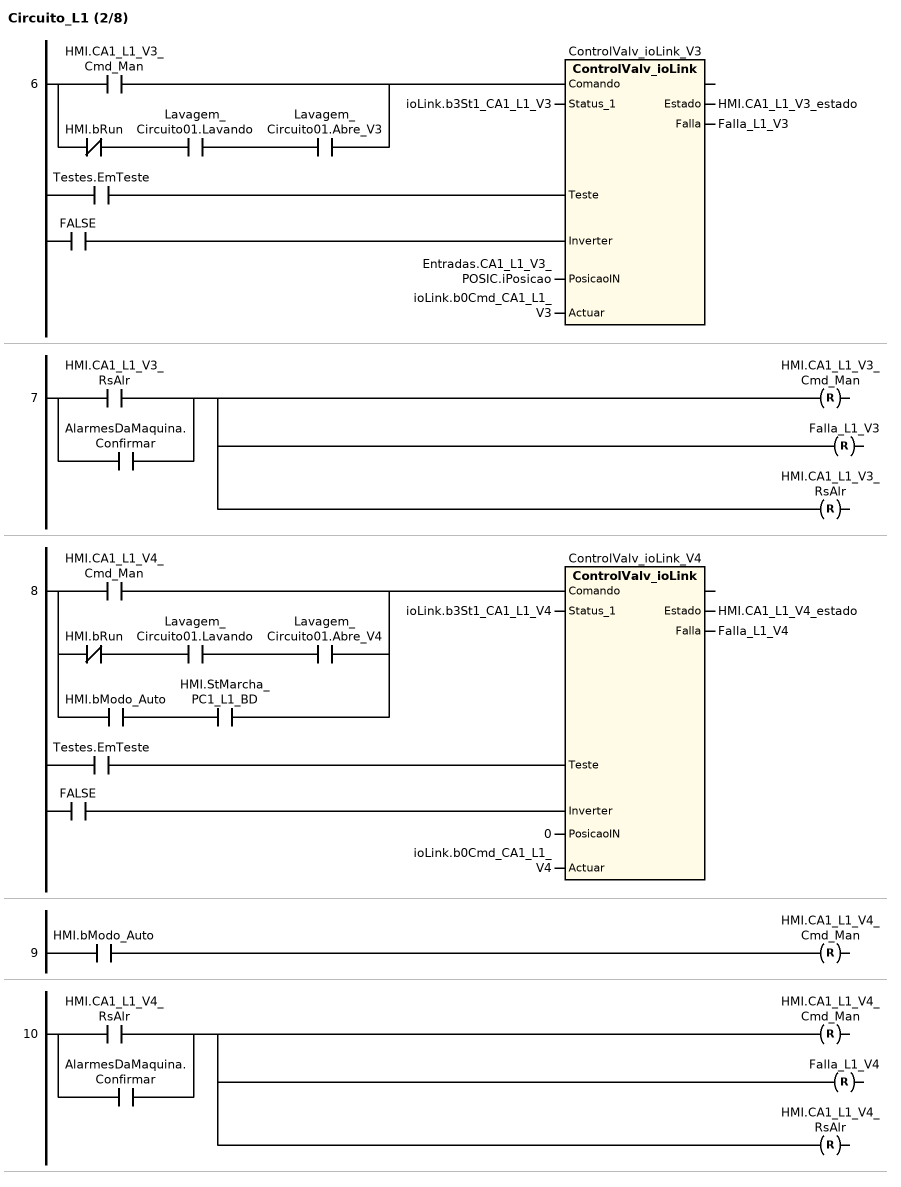
// NETWORK 6
ControlValv_ioLink_V3(
    Comando := HMI.CA1_L1_V3_Cmd_Man OR NOT HMI.bRun AND Lavagem_Circuito01.Lavando AND Lavagem_Circuito01.Abre_V3,
    Status_1 := ioLink.b3St1_CA1_L1_V3,
    Teste := Testes.EmTeste,
    Inverter := FALSE,
    PosicaoIN := Entradas.CA1_L1_V3_POSIC.iPosicao,
    Actuar := ioLink.b0Cmd_CA1_L1_V3,
    Estado => HMI.CA1_L1_V3_estado,
    Falla => Falla_L1_V3); // ControlValv_ioLink

// NETWORK 7
_w3 := HMI.CA1_L1_V3_RsAlr OR AlarmesDaMaquina.Confirmar;
HMI.CA1_L1_V3_Cmd_Man R= _w3;
Falla_L1_V3 R= _w3;
HMI.CA1_L1_V3_RsAlr R= _w3;

// NETWORK 8
ControlValv_ioLink_V4(
    Comando := HMI.CA1_L1_V4_Cmd_Man OR NOT HMI.bRun AND Lavagem_Circuito01.Lavando AND Lavagem_Circuito01.Abre_V4 OR HMI.bModo_Auto AND HMI.StMarcha_PC1_L1_BD,
    Status_1 := ioLink.b3St1_CA1_L1_V4,
    Teste := Testes.EmTeste,
    Inverter := FALSE,
    PosicaoIN := 0,
    Actuar := ioLink.b0Cmd_CA1_L1_V4,
    Estado => HMI.CA1_L1_V4_estado,
    Falla => Falla_L1_V4); // ControlValv_ioLink

// NETWORK 9
HMI.CA1_L1_V4_Cmd_Man R= HMI.bModo_Auto;

// NETWORK 10
_w4 := HMI.CA1_L1_V4_RsAlr OR AlarmesDaMaquina.Confirmar;
HMI.CA1_L1_V4_Cmd_Man R= _w4;
Falla_L1_V4 R= _w4;
HMI.CA1_L1_V4_RsAlr R= _w4;

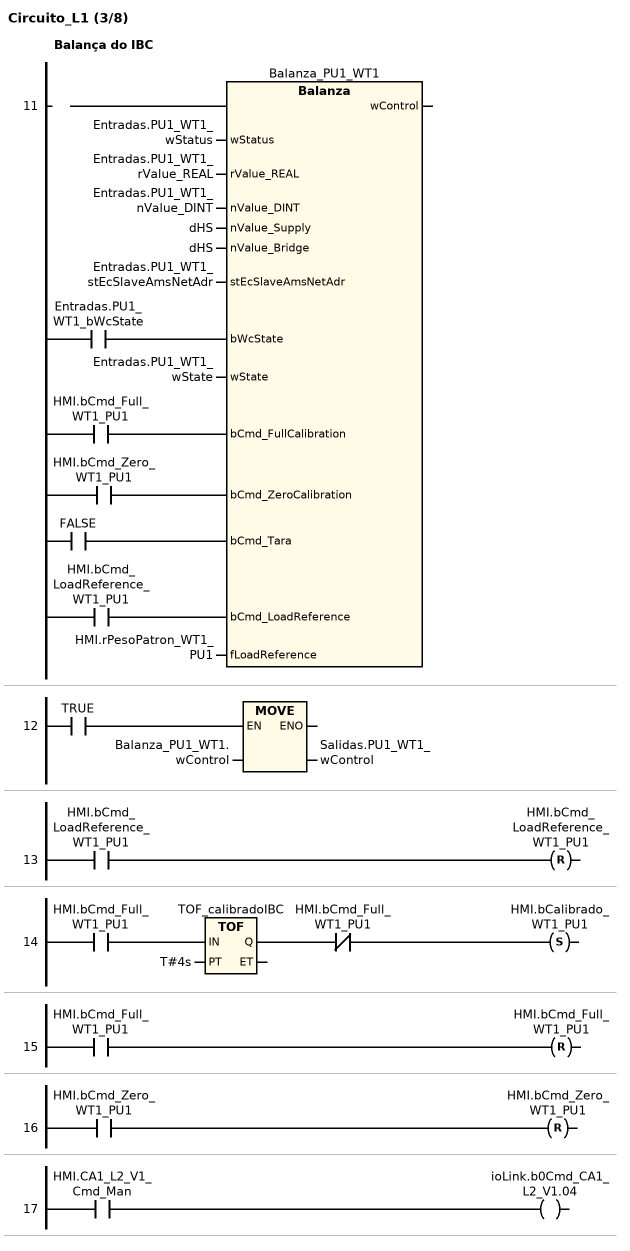
// NETWORK 11: Balança do IBC
Balanza_PU1_WT1(
    wStatus := Entradas.PU1_WT1_wStatus,
    rValue_REAL := Entradas.PU1_WT1_rValue_REAL,
    nValue_DINT := Entradas.PU1_WT1_nValue_DINT,
    nValue_Supply := dHS,
    nValue_Bridge := dHS,
    stEcSlaveAmsNetAdr := Entradas.PU1_WT1_stEcSlaveAmsNetAdr,
    bWcState := Entradas.PU1_WT1_bWcState,
    wState := Entradas.PU1_WT1_wState,
    bCmd_FullCalibration := HMI.bCmd_Full_WT1_PU1,
    bCmd_ZeroCalibration := HMI.bCmd_Zero_WT1_PU1,
    bCmd_Tara := FALSE,
    bCmd_LoadReference := HMI.bCmd_LoadReference_WT1_PU1,
    fLoadReference := HMI.rPesoPatron_WT1_PU1); // Balanza

// NETWORK 12
Salidas.PU1_WT1_wControl := Balanza_PU1_WT1.wControl;

// NETWORK 13
HMI.bCmd_LoadReference_WT1_PU1 R= HMI.bCmd_LoadReference_WT1_PU1;

// NETWORK 14
TOF_calibradoIBC(IN := HMI.bCmd_Full_WT1_PU1, PT := T#4s); // TOF
HMI.bCalibrado_WT1_PU1 S= TOF_calibradoIBC.Q AND NOT HMI.bCmd_Full_WT1_PU1;

// NETWORK 15
HMI.bCmd_Full_WT1_PU1 R= HMI.bCmd_Full_WT1_PU1;

// NETWORK 16
HMI.bCmd_Zero_WT1_PU1 R= HMI.bCmd_Zero_WT1_PU1;

// NETWORK 17
ioLink.b0Cmd_CA1_L2_V1.04 := HMI.CA1_L2_V1_Cmd_Man;

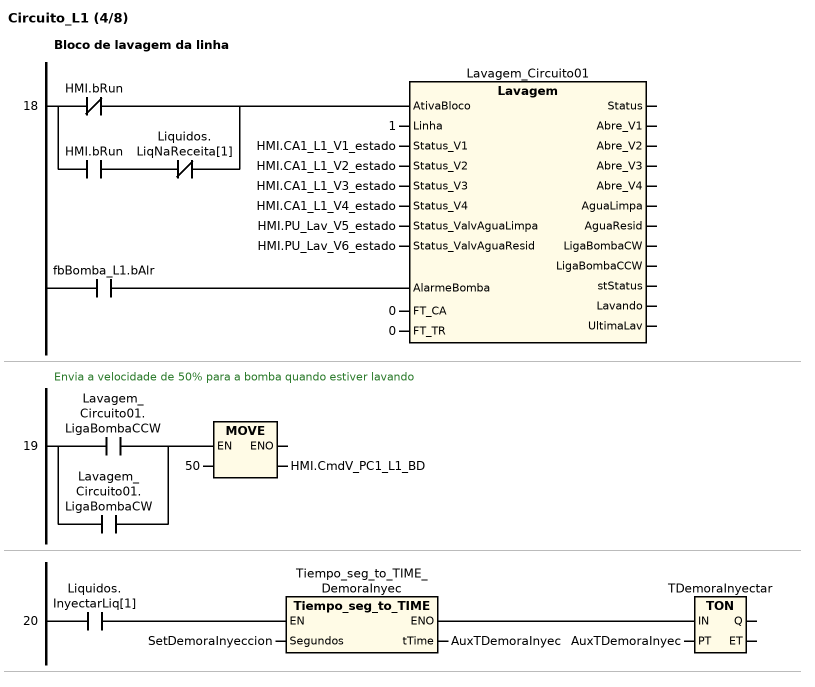
// NETWORK 18: Bloco de lavagem da linha
Lavagem_Circuito01(
    AtivaBloco := NOT HMI.bRun OR HMI.bRun AND NOT Liquidos.LiqNaReceita[1],
    Linha := 1,
    Status_V1 := HMI.CA1_L1_V1_estado,
    Status_V2 := HMI.CA1_L1_V2_estado,
    Status_V3 := HMI.CA1_L1_V3_estado,
    Status_V4 := HMI.CA1_L1_V4_estado,
    Status_ValvAguaLimpa := HMI.PU_Lav_V5_estado,
    Status_ValvAguaResid := HMI.PU_Lav_V6_estado,
    AlarmeBomba := fbBomba_L1.bAlr,
    FT_CA := 0,
    FT_TR := 0); // Lavagem

// NETWORK 19
// Envia a velocidade de 50% para a bomba quando estiver lavando
IF Lavagem_Circuito01.LigaBombaCCW OR Lavagem_Circuito01.LigaBombaCW THEN HMI.CmdV_PC1_L1_BD := 50; END_IF

// NETWORK 20
_w5 := Liquidos.InyectarLiq[1];
IF _w5 THEN
    Tiempo_seg_to_TIME_DemoraInyec(Segundos := SetDemoraInyeccion, tTime => AuxTDemoraInyec); // Tiempo_seg_to_TIME
END_IF
TDemoraInyectar(IN := _w5, PT := AuxTDemoraInyec); // TON

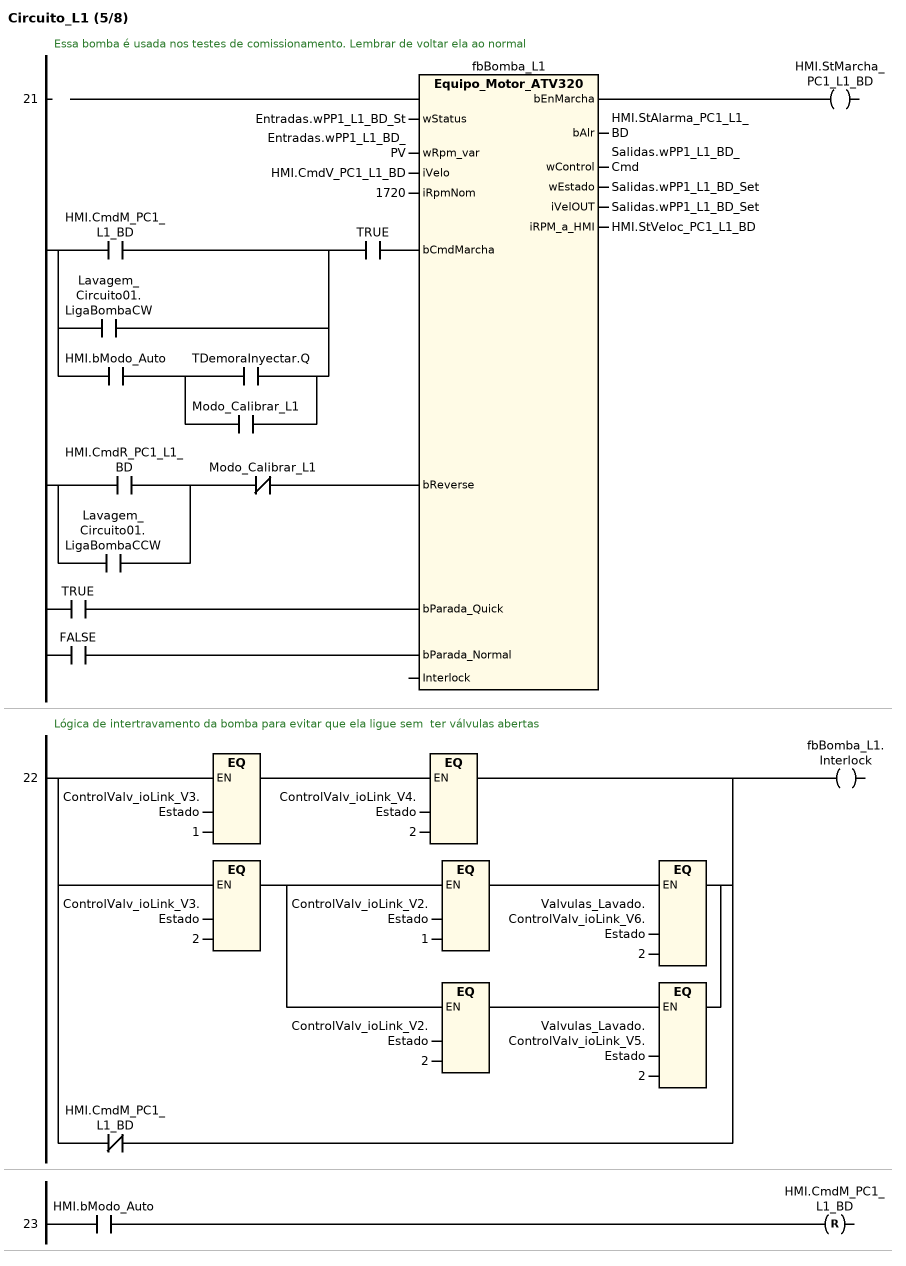
// NETWORK 21
// Essa bomba é usada nos testes de comissionamento. Lembrar de voltar ela ao normal
fbBomba_L1(
    wStatus := Entradas.wPP1_L1_BD_St,
    wRpm_var := Entradas.wPP1_L1_BD_PV,
    iVelo := HMI.CmdV_PC1_L1_BD,
    iRpmNom := 1720,
    bCmdMarcha := (HMI.CmdM_PC1_L1_BD OR Lavagem_Circuito01.LigaBombaCW OR HMI.bModo_Auto AND (TDemoraInyectar.Q OR Modo_Calibrar_L1)) AND TRUE,
    bReverse := (HMI.CmdR_PC1_L1_BD OR Lavagem_Circuito01.LigaBombaCCW) AND NOT Modo_Calibrar_L1,
    bParada_Quick := TRUE,
    bParada_Normal := FALSE,
    bAlr => HMI.StAlarma_PC1_L1_BD,
    wControl => Salidas.wPP1_L1_BD_Cmd,
    wEstado => Salidas.wPP1_L1_BD_Set,
    iVelOUT => Salidas.wPP1_L1_BD_Set,
    iRPM_a_HMI => HMI.StVeloc_PC1_L1_BD); // Equipo_Motor_ATV320
HMI.StMarcha_PC1_L1_BD := fbBomba_L1.bEnMarcha;

// NETWORK 22
// Lógica de intertravamento da bomba para evitar que ela ligue sem  ter válvulas abertas
_w6 := NOT HMI.CmdM_PC1_L1_BD;
IF NOT _w6 THEN
    _w7 := ControlValv_ioLink_V3.Estado = 2;
    _w6 := ControlValv_ioLink_V3.Estado = 1 AND ControlValv_ioLink_V4.Estado = 2 OR (_w7 AND ControlValv_ioLink_V2.Estado = 1 AND Valvulas_Lavado.ControlValv_ioLink_V6.Estado = 2 OR _w7 AND ControlValv_ioLink_V2.Estado = 2 AND Valvulas_Lavado.ControlValv_ioLink_V5.Estado = 2);
END_IF
fbBomba_L1.Interlock := _w6;

// NETWORK 23
HMI.CmdM_PC1_L1_BD R= HMI.bModo_Auto;

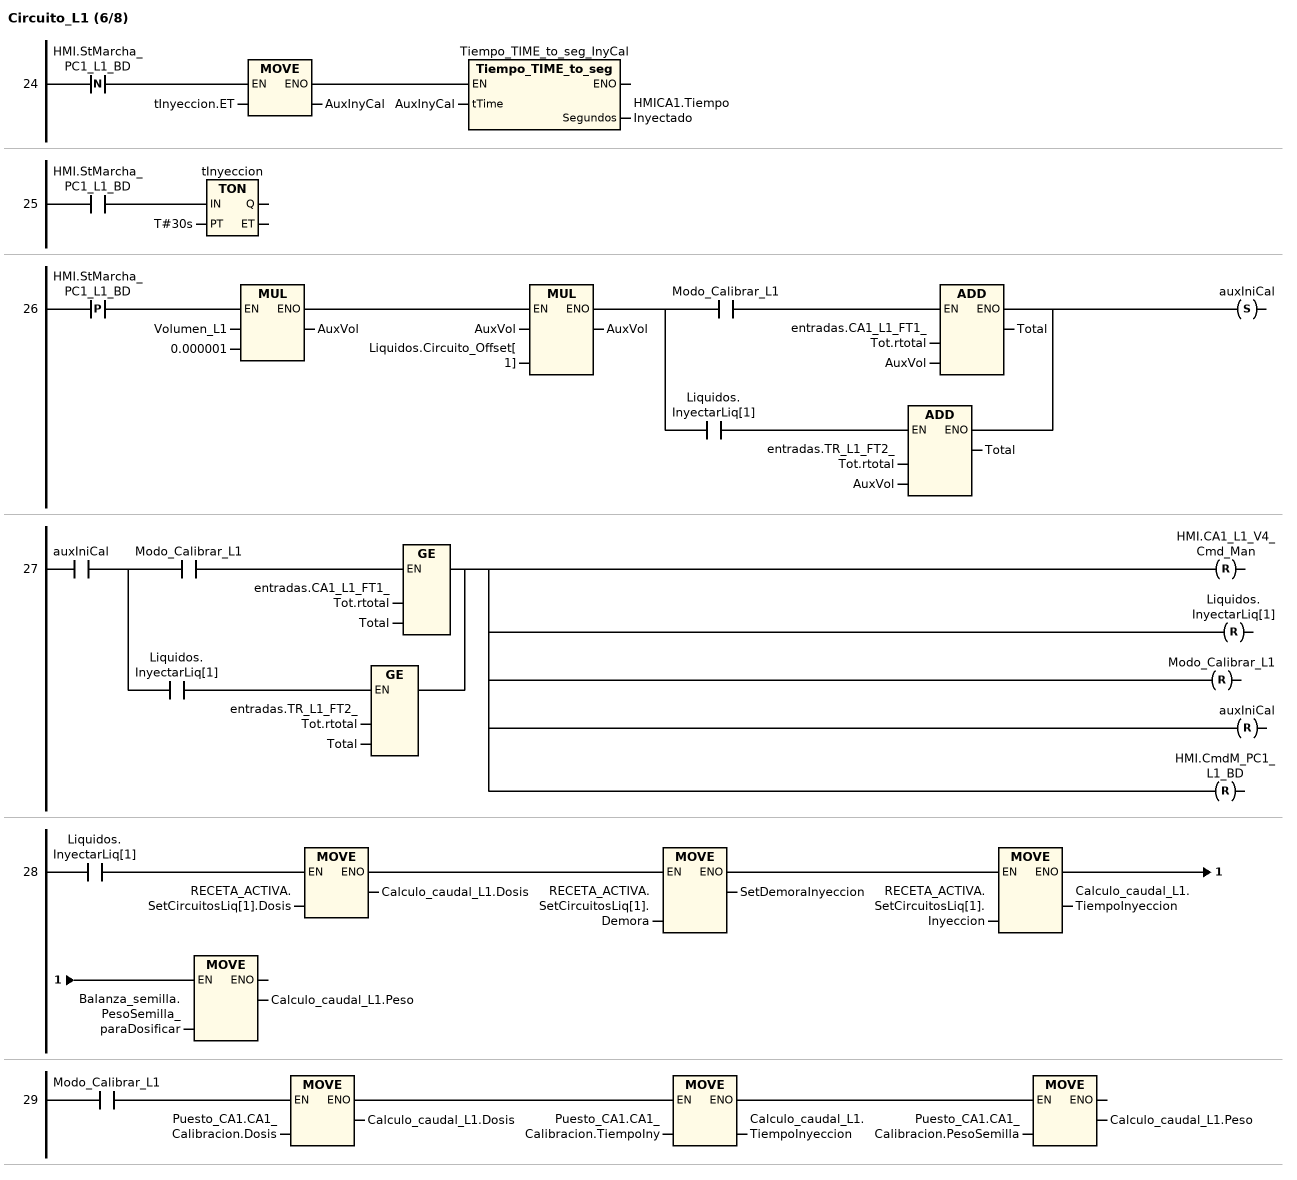
// NETWORK 24
_ft1(CLK := HMI.StMarcha_PC1_L1_BD);
_w8 := _ft1.Q;
IF _w8 THEN AuxInyCal := tInyeccion.ET; END_IF
IF _w8 THEN
    Tiempo_TIME_to_seg_InyCal(tTime := AuxInyCal, Segundos => HMICA1.TiempoInyectado); // Tiempo_TIME_to_seg
END_IF

// NETWORK 25
tInyeccion(IN := HMI.StMarcha_PC1_L1_BD, PT := T#30s); // TON

// NETWORK 26
_rt1(CLK := HMI.StMarcha_PC1_L1_BD);
_w9 := _rt1.Q;
IF _w9 THEN AuxVol := Volumen_L1 * 0.000001; END_IF
IF _w9 THEN AuxVol := AuxVol * Liquidos.Circuito_Offset[1]; END_IF
IF _w9 AND Modo_Calibrar_L1 THEN Total := entradas.CA1_L1_FT1_Tot.rtotal + AuxVol; END_IF
IF _w9 AND Liquidos.InyectarLiq[1] THEN Total := entradas.TR_L1_FT2_Tot.rtotal + AuxVol; END_IF
auxIniCal S= _w9 AND Modo_Calibrar_L1 OR _w9 AND Liquidos.InyectarLiq[1];

// NETWORK 27
_w10 := auxIniCal AND Modo_Calibrar_L1 AND entradas.CA1_L1_FT1_Tot.rtotal >= Total OR auxIniCal AND Liquidos.InyectarLiq[1] AND entradas.TR_L1_FT2_Tot.rtotal >= Total;
HMI.CA1_L1_V4_Cmd_Man R= _w10;
Liquidos.InyectarLiq[1] R= _w10;
Modo_Calibrar_L1 R= _w10;
auxIniCal R= _w10;
HMI.CmdM_PC1_L1_BD R= _w10;

// NETWORK 28
_w11 := Liquidos.InyectarLiq[1];
IF _w11 THEN Calculo_caudal_L1.Dosis := RECETA_ACTIVA.SetCircuitosLiq[1].Dosis; END_IF
IF _w11 THEN SetDemoraInyeccion := RECETA_ACTIVA.SetCircuitosLiq[1].Demora; END_IF
IF _w11 THEN Calculo_caudal_L1.TiempoInyeccion := RECETA_ACTIVA.SetCircuitosLiq[1].Inyeccion; END_IF
IF _w11 THEN Calculo_caudal_L1.Peso := Balanza_semilla.PesoSemilla_paraDosificar; END_IF

// NETWORK 29
_w12 := Modo_Calibrar_L1;
IF _w12 THEN Calculo_caudal_L1.Dosis := Puesto_CA1.CA1_Calibracion.Dosis; END_IF
IF _w12 THEN Calculo_caudal_L1.TiempoInyeccion := Puesto_CA1.CA1_Calibracion.TiempoIny; END_IF
IF _w12 THEN Calculo_caudal_L1.Peso := Puesto_CA1.CA1_Calibracion.PesoSemilla; END_IF

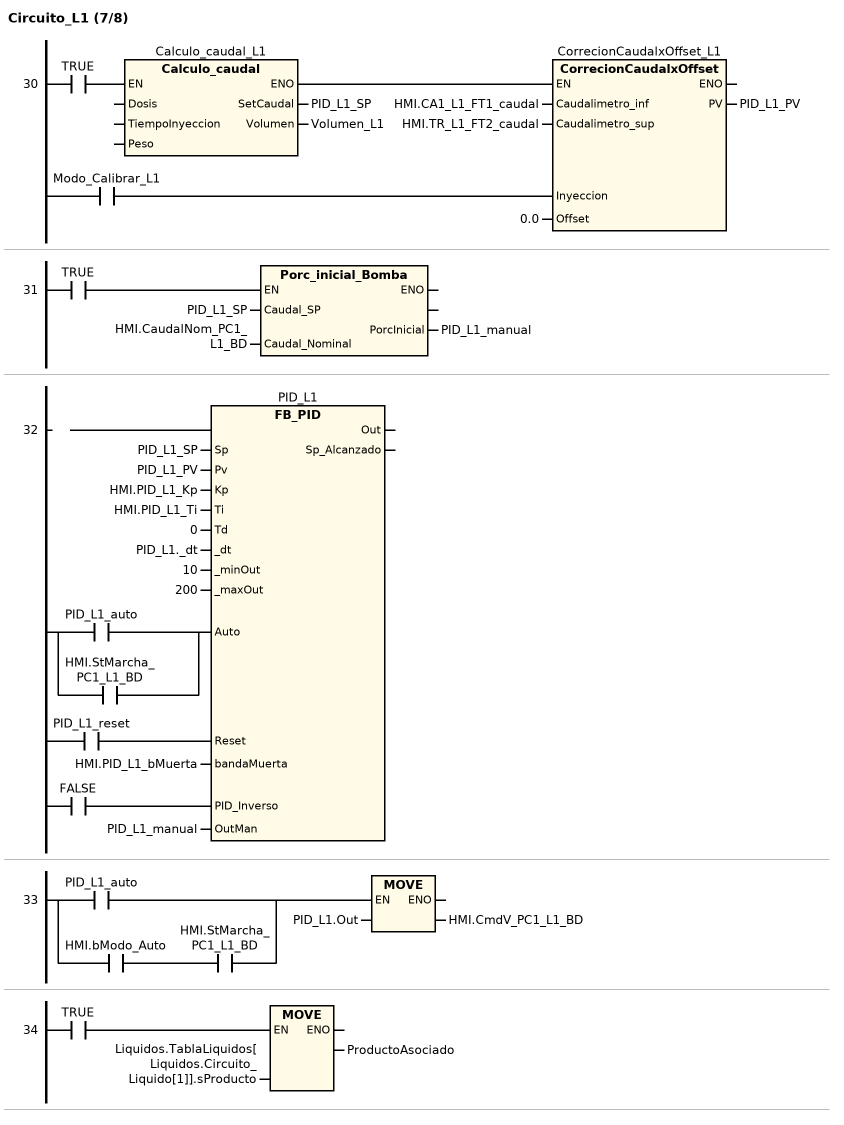
// NETWORK 30
Calculo_caudal_L1(SetCaudal => PID_L1_SP, Volumen => Volumen_L1); // Calculo_caudal
CorrecionCaudalxOffset_L1(
    Caudalimetro_inf := HMI.CA1_L1_FT1_caudal,
    Caudalimetro_sup := HMI.TR_L1_FT2_caudal,
    Inyeccion := Modo_Calibrar_L1,
    Offset := 0.0,
    PV => PID_L1_PV); // CorrecionCaudalxOffset

// NETWORK 31
Porc_inicial_Bomba(Caudal_SP := PID_L1_SP, Caudal_Nominal := HMI.CaudalNom_PC1_L1_BD, PorcInicial => PID_L1_manual);

// NETWORK 32
PID_L1(
    Sp := PID_L1_SP,
    Pv := PID_L1_PV,
    Kp := HMI.PID_L1_Kp,
    Ti := HMI.PID_L1_Ti,
    Td := 0,
    _dt := PID_L1._dt,
    _minOut := 10,
    _maxOut := 200,
    Auto := PID_L1_auto OR HMI.StMarcha_PC1_L1_BD,
    Reset := PID_L1_reset,
    bandaMuerta := HMI.PID_L1_bMuerta,
    PID_Inverso := FALSE,
    OutMan := PID_L1_manual); // FB_PID

// NETWORK 33
IF PID_L1_auto OR HMI.bModo_Auto AND HMI.StMarcha_PC1_L1_BD THEN HMI.CmdV_PC1_L1_BD := PID_L1.Out; END_IF

// NETWORK 34
ProductoAsociado := Liquidos.TablaLiquidos[Liquidos.Circuito_Liquido[1]].sProducto;

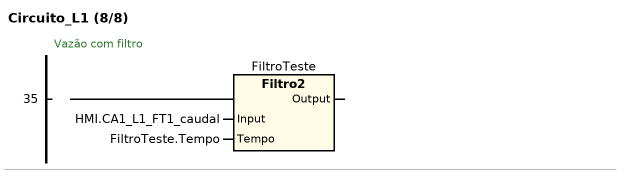
// NETWORK 35
// Vazão com filtro
FiltroTeste(Input := HMI.CA1_L1_FT1_caudal, Tempo := FiltroTeste.Tempo); // Filtro2

END_PROGRAM

// ---- POUs/Secuencias/LavadoCircuitoLiquidos.TcPOU
FUNCTION_BLOCK LavadoCircuitoLiquidos
VAR_INPUT
	bModoEco:BOOL;
	rCaudalLlenado:REAL;
	rCaudalVaciado:REAL;
	bBomba_enMarcha:BOOL;
	rVelocBombaVaciado:REAL;
	rVelocBombaLavado:REAL;
	tSetTmrVaciado:TIME;
	tSetTmrLlenado:TIME;
	iCantCiclosECO:INT;
	iCantCiclosLavado:INT;
	wEstadoV_AguaResidual:WORD;//bit1=cerrada  bit0=abierta
	wEstadoV_Agua:WORD;//bit1=cerrada  bit0=abierta
	wEstadoCal_V1:WORD;//bit1=a inyeccion  bit0=a probeta
	wEstadoV1:WORD;//bit1=cerrada  bit0=abierta
	wEstadoV2:WORD;//bit1=a proceso  bit0=a limpieza
	wEstadoV3:WORD;//bit1=a agua  bit0=a agua residual
	
END_VAR
VAR_OUTPUT
	rPorcCiclosECO:REAL;
	rPorcCiclosLavado:REAL;
	rPorcAvance:REAL;
	bCa_V1_aProbeta:BOOL;
	bV1_Abrir:BOOL;
	bV2_aLimpieza:BOOL;
	bV3_aResidual:BOOL;
	bV_Residual:BOOL;
	bV_Agua:BOOL;
	rSetVelocBomba:REAL;
	bMarchaBomba:BOOL;
	bReverseBomba:BOOL;

	
END_VAR
VAR_IN_OUT
	bInicioLavado:BOOL;	
	bCancelar:BOOL;
END_VAR
VAR
	TON_Vaciado: TON;
	FinVaciado:BOOL;
	VaciarCircuito:BOOL;
	FinLlenado:BOOL;
	LlenarCircuito:BOOL;
	LavadoLlenar:BOOL;
	LavadoVaciar:BOOL;
	TON_Llenado: TON;
	BombaForward:BOOL;
	BombaReverse:BOOL;
	CtrCiclosModoECO:INT;
	CtrCiclosLavado:INT;
	SetTotalCiclos:REAL;
	TotalCiclosActual:INT;
	rAux:REAL;
	TON_llenadoProbeta: TON;
	TON_vaciadoProbeta: TON;
END_VAR
VAR // added by the converter: edge detectors and wires of the graphical bodies
    _rt1, _rt2 : R_TRIG;
    _w1, _w2, _w3, _w4, _w5, _w6, _w7, _w8 : BOOL;
END_VAR

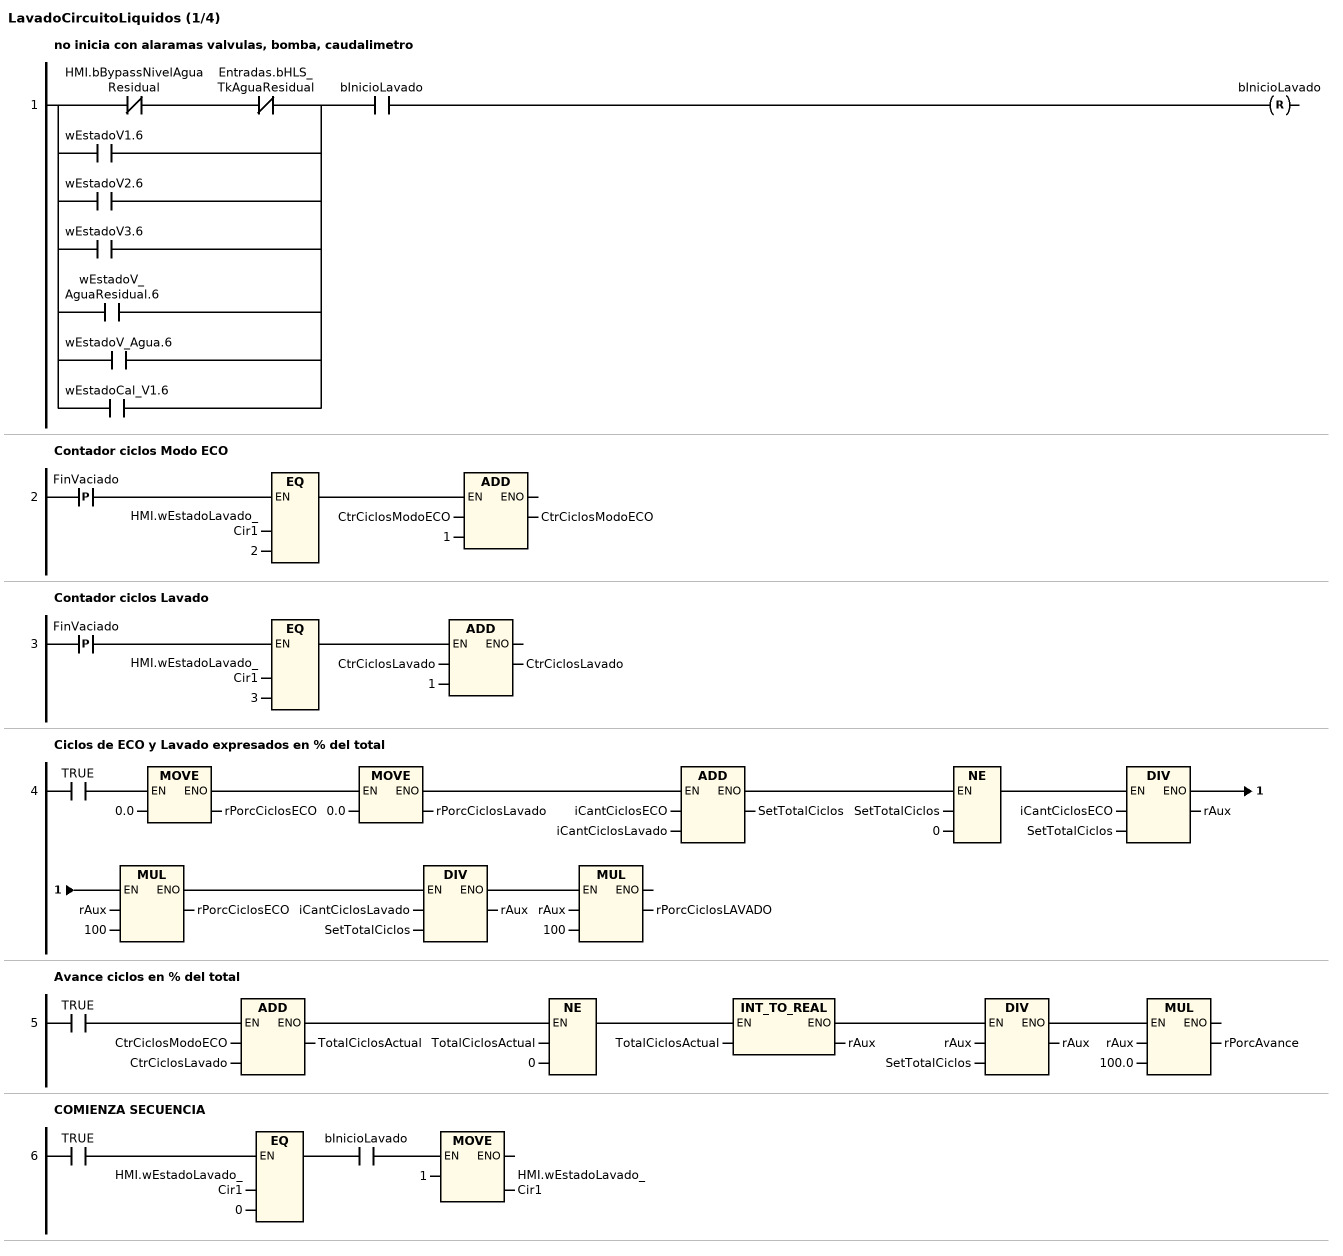
// NETWORK 1: no inicia con alaramas valvulas, bomba, caudalimetro
bInicioLavado R= (NOT HMI.bBypassNivelAguaResidual AND NOT Entradas.bHLS_TkAguaResidual OR wEstadoV1.6 OR wEstadoV2.6 OR wEstadoV3.6 OR wEstadoV_AguaResidual.6 OR wEstadoV_Agua.6 OR wEstadoCal_V1.6) AND bInicioLavado;

// NETWORK 2: Contador ciclos Modo ECO
_rt1(CLK := FinVaciado);
IF _rt1.Q AND HMI.wEstadoLavado_Cir1 = 2 THEN CtrCiclosModoECO := CtrCiclosModoECO + 1; END_IF

// NETWORK 3: Contador ciclos Lavado
_rt2(CLK := FinVaciado);
IF _rt2.Q AND HMI.wEstadoLavado_Cir1 = 3 THEN CtrCiclosLavado := CtrCiclosLavado + 1; END_IF

// NETWORK 4: Ciclos de ECO y Lavado expresados en % del total
rPorcCiclosECO := 0.0;
rPorcCiclosLavado := 0.0;
SetTotalCiclos := iCantCiclosECO + iCantCiclosLavado;
_w1 := SetTotalCiclos <> 0;
IF _w1 THEN rAux := iCantCiclosECO / SetTotalCiclos; END_IF
IF _w1 THEN rPorcCiclosECO := rAux * 100; END_IF
IF _w1 THEN rAux := iCantCiclosLavado / SetTotalCiclos; END_IF
IF _w1 THEN rPorcCiclosLAVADO := rAux * 100; END_IF

// NETWORK 5: Avance ciclos en % del total
TotalCiclosActual := CtrCiclosModoECO + CtrCiclosLavado;
_w2 := TotalCiclosActual <> 0;
IF _w2 THEN rAux := INT_TO_REAL(TotalCiclosActual); END_IF
IF _w2 THEN rAux := rAux / SetTotalCiclos; END_IF
IF _w2 THEN rPorcAvance := rAux * 100.0; END_IF

// NETWORK 6: COMIENZA SECUENCIA
IF HMI.wEstadoLavado_Cir1 = 0 AND bInicioLavado THEN HMI.wEstadoLavado_Cir1 := 1; END_IF

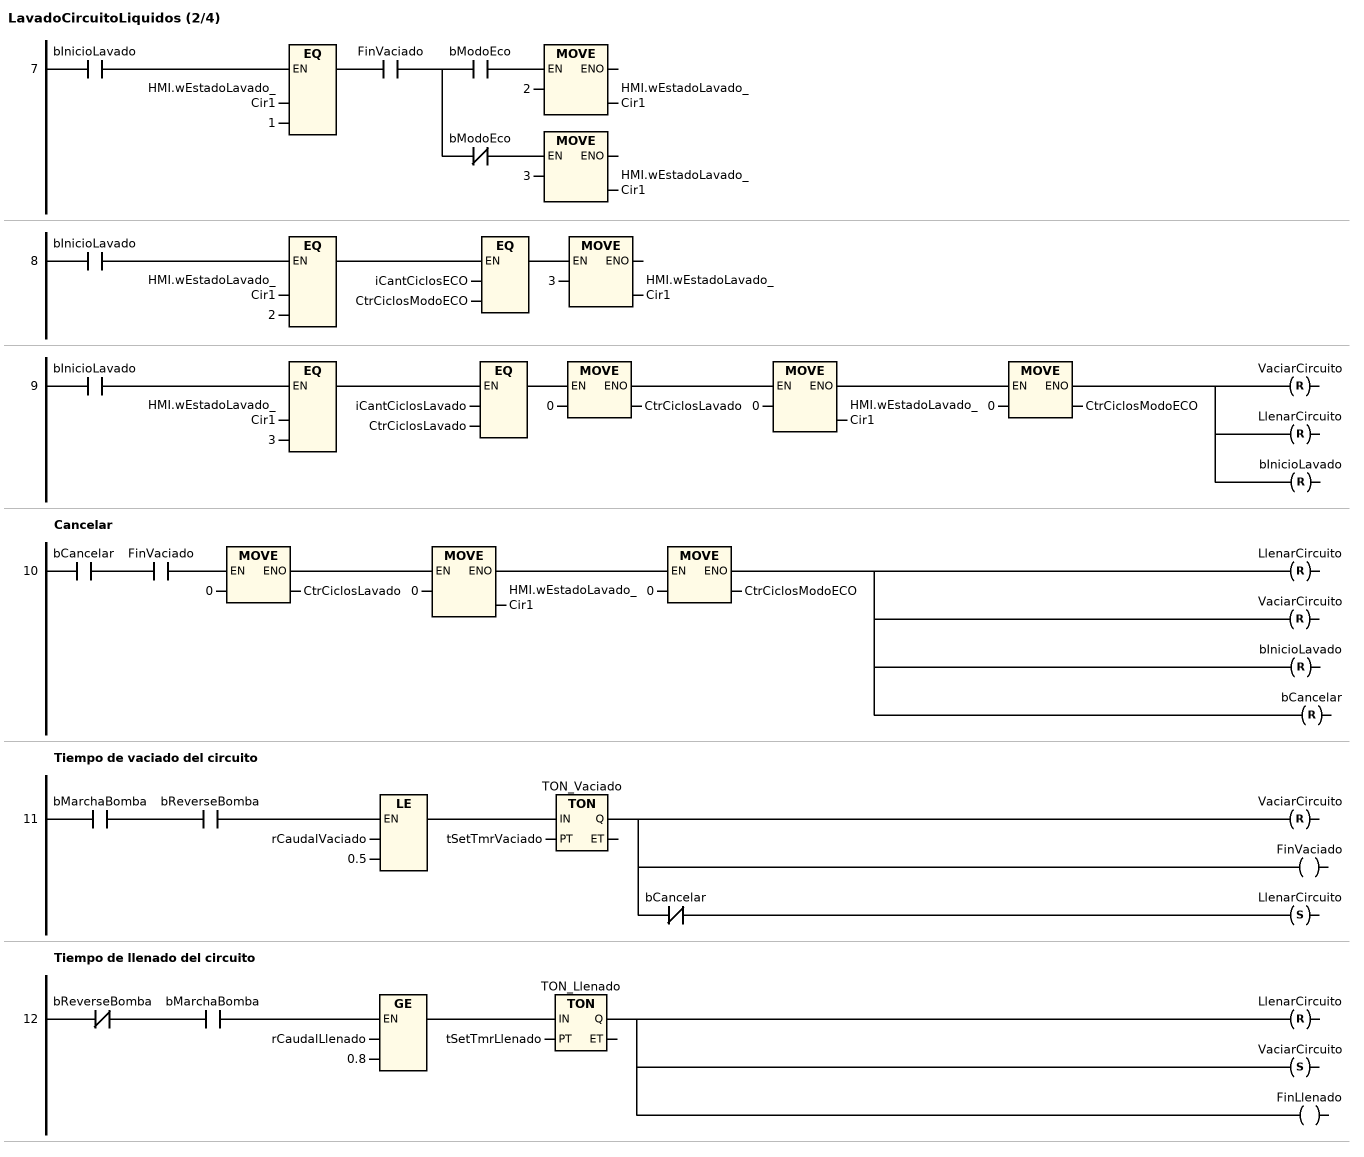
// NETWORK 7
_w3 := (bInicioLavado AND HMI.wEstadoLavado_Cir1 = 1) AND FinVaciado;
IF _w3 AND bModoEco THEN HMI.wEstadoLavado_Cir1 := 2; END_IF
IF _w3 AND NOT bModoEco THEN HMI.wEstadoLavado_Cir1 := 3; END_IF

// NETWORK 8
IF bInicioLavado AND HMI.wEstadoLavado_Cir1 = 2 AND iCantCiclosECO = CtrCiclosModoECO THEN
    HMI.wEstadoLavado_Cir1 := 3;
END_IF

// NETWORK 9
_w4 := bInicioLavado AND HMI.wEstadoLavado_Cir1 = 3 AND iCantCiclosLavado = CtrCiclosLavado;
IF _w4 THEN CtrCiclosLavado := 0; END_IF
IF _w4 THEN HMI.wEstadoLavado_Cir1 := 0; END_IF
IF _w4 THEN CtrCiclosModoECO := 0; END_IF
VaciarCircuito R= _w4;
LlenarCircuito R= _w4;
bInicioLavado R= _w4;

// NETWORK 10: Cancelar
_w5 := bCancelar AND FinVaciado;
IF _w5 THEN CtrCiclosLavado := 0; END_IF
IF _w5 THEN HMI.wEstadoLavado_Cir1 := 0; END_IF
IF _w5 THEN CtrCiclosModoECO := 0; END_IF
LlenarCircuito R= _w5;
VaciarCircuito R= _w5;
bInicioLavado R= _w5;
bCancelar R= _w5;

// NETWORK 11: Tiempo de vaciado del circuito
TON_Vaciado(IN := bMarchaBomba AND bReverseBomba AND rCaudalVaciado <= 0.5, PT := tSetTmrVaciado); // TON
VaciarCircuito R= TON_Vaciado.Q;
FinVaciado := TON_Vaciado.Q;
LlenarCircuito S= TON_Vaciado.Q AND NOT bCancelar;

// NETWORK 12: Tiempo de llenado del circuito
TON_Llenado(IN := NOT bReverseBomba AND bMarchaBomba AND rCaudalLlenado >= 0.8, PT := tSetTmrLlenado); // TON
LlenarCircuito R= TON_Llenado.Q;
VaciarCircuito S= TON_Llenado.Q;
FinLlenado := TON_Llenado.Q;

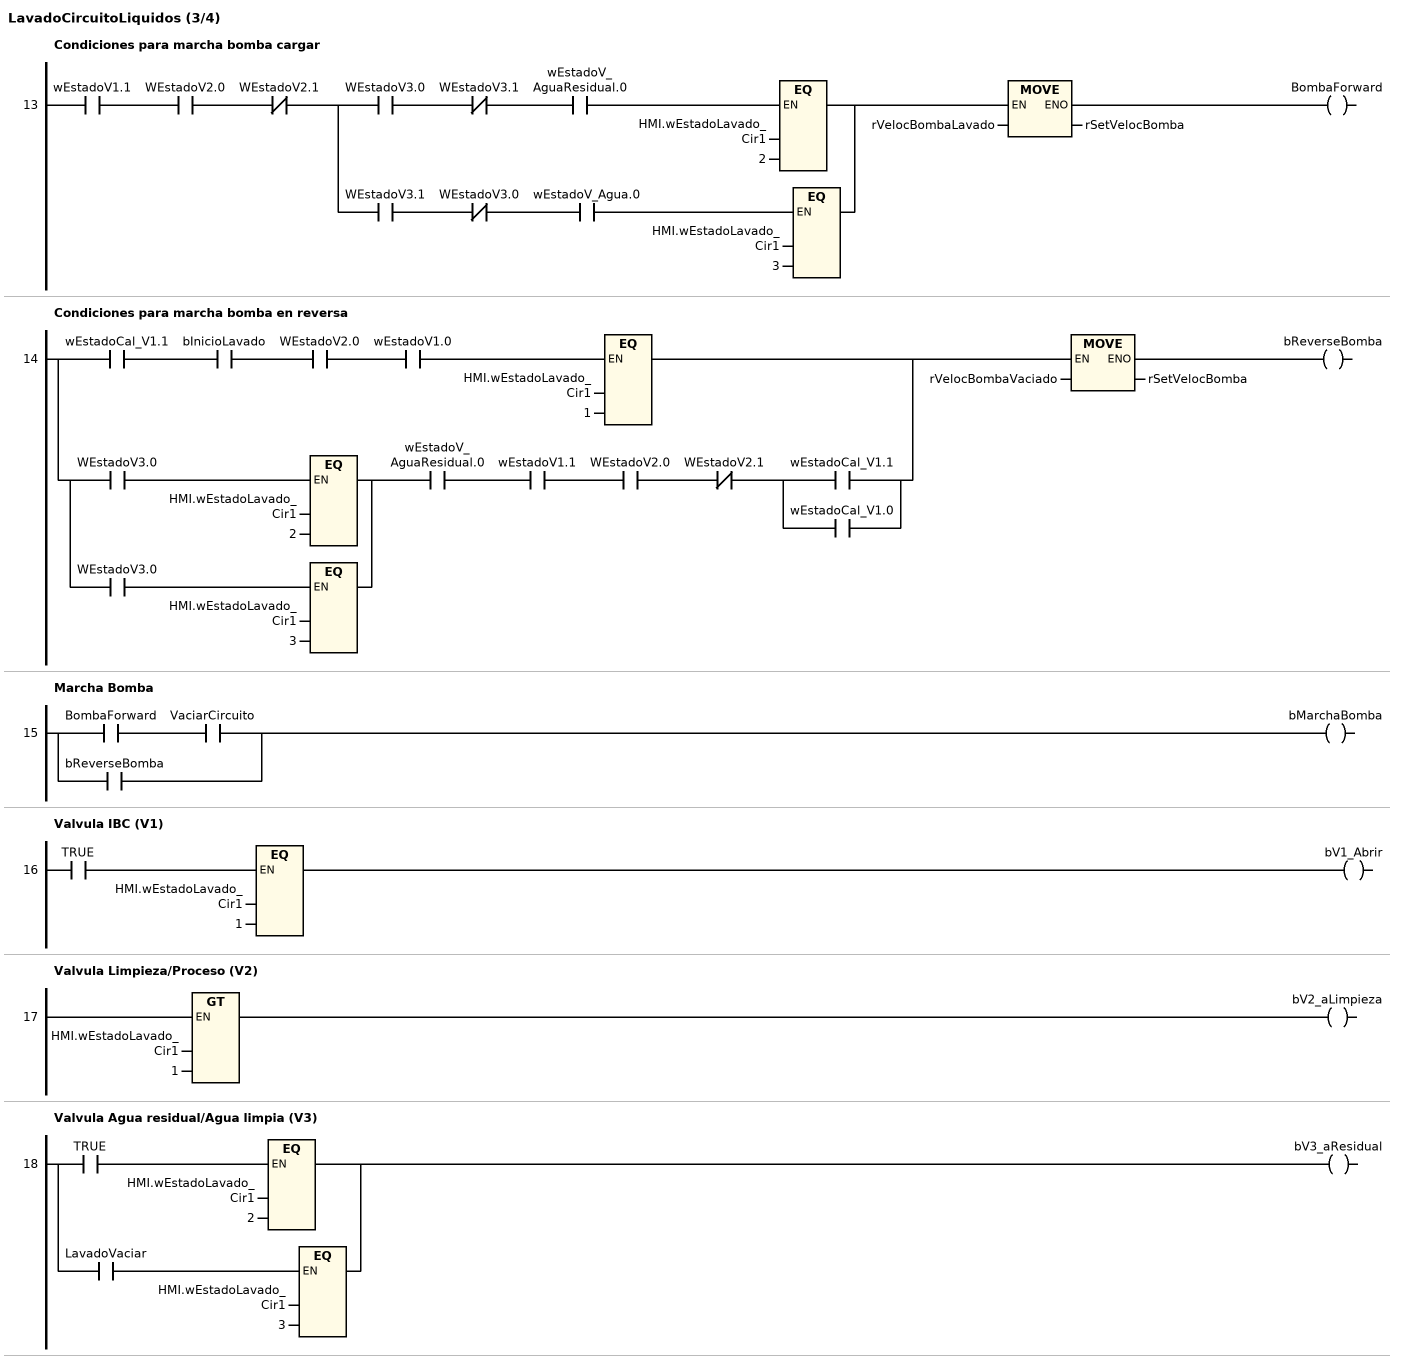
// NETWORK 13: Condiciones para marcha bomba cargar
_w6 := wEstadoV1.1 AND WEstadoV2.0 AND NOT WEstadoV2.1;
_w7 := (_w6 AND WEstadoV3.0) AND NOT WEstadoV3.1 AND wEstadoV_AguaResidual.0 AND HMI.wEstadoLavado_Cir1 = 2 OR (_w6 AND WEstadoV3.1) AND NOT WEstadoV3.0 AND wEstadoV_Agua.0 AND HMI.wEstadoLavado_Cir1 = 3;
IF _w7 THEN rSetVelocBomba := rVelocBombaLavado; END_IF
BombaForward := _w7;

// NETWORK 14: Condiciones para marcha bomba en reversa
_w8 := wEstadoCal_V1.1 AND bInicioLavado AND WEstadoV2.0 AND wEstadoV1.0 AND HMI.wEstadoLavado_Cir1 = 1 OR (WEstadoV3.0 AND HMI.wEstadoLavado_Cir1 = 2 OR WEstadoV3.0 AND HMI.wEstadoLavado_Cir1 = 3) AND wEstadoV_AguaResidual.0 AND wEstadoV1.1 AND WEstadoV2.0 AND NOT WEstadoV2.1 AND (wEstadoCal_V1.1 OR wEstadoCal_V1.0);
IF _w8 THEN rSetVelocBomba := rVelocBombaVaciado; END_IF
bReverseBomba := _w8;

// NETWORK 15: Marcha Bomba
bMarchaBomba := BombaForward AND VaciarCircuito OR bReverseBomba;

// NETWORK 16: Valvula IBC (V1)
bV1_Abrir := HMI.wEstadoLavado_Cir1 = 1;

// NETWORK 17: Valvula Limpieza/Proceso (V2)
bV2_aLimpieza := HMI.wEstadoLavado_Cir1 > 1;

// NETWORK 18: Valvula Agua residual/Agua limpia (V3)
bV3_aResidual := HMI.wEstadoLavado_Cir1 = 2 OR LavadoVaciar AND HMI.wEstadoLavado_Cir1 = 3;

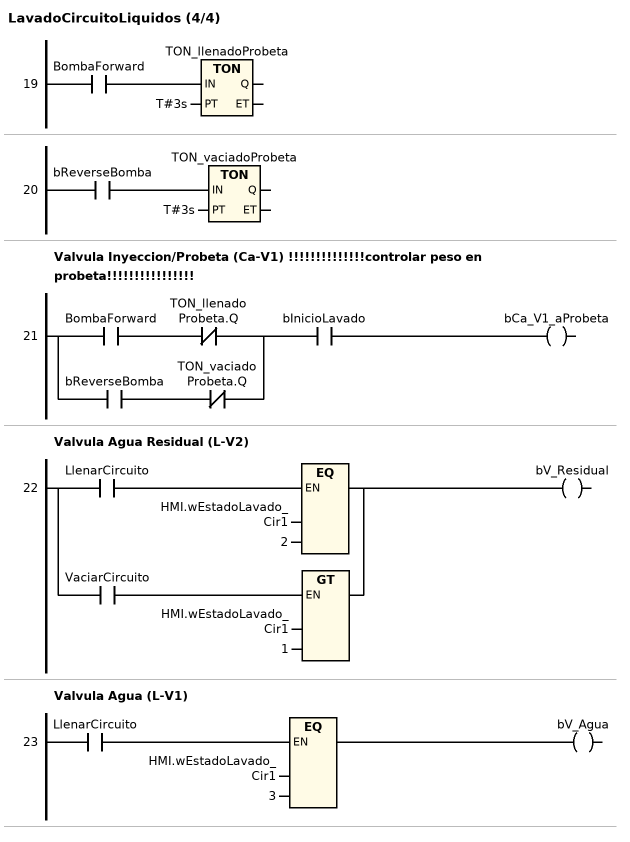
// NETWORK 19
TON_llenadoProbeta(IN := BombaForward, PT := T#3s); // TON

// NETWORK 20
TON_vaciadoProbeta(IN := bReverseBomba, PT := T#3s); // TON

// NETWORK 21: Valvula Inyeccion/Probeta (Ca-V1) !!!!!!!!!!!!!!controlar peso en probeta!!!!!!!!!!!!!!!!
bCa_V1_aProbeta := (BombaForward AND NOT TON_llenadoProbeta.Q OR bReverseBomba AND NOT TON_vaciadoProbeta.Q) AND bInicioLavado;

// NETWORK 22: Valvula Agua Residual (L-V2)
bV_Residual := LlenarCircuito AND HMI.wEstadoLavado_Cir1 = 2 OR VaciarCircuito AND HMI.wEstadoLavado_Cir1 > 1;

// NETWORK 23: Valvula Agua (L-V1)
bV_Agua := LlenarCircuito AND HMI.wEstadoLavado_Cir1 = 3;

END_FUNCTION_BLOCK

// ---- POUs/Secuencias/Totalizador.TcPOU
FUNCTION_BLOCK Totalizador
VAR_INPUT
	PV:	REAL;
	Medir: BOOL;
END_VAR
VAR_OUTPUT
	Volumen: REAL;
END_VAR
VAR_IN_OUT
	Reset:BOOL;
END_VAR	
VAR
	fbMuestra: TON;
END_VAR

fbMuestra(IN:=(Medir AND NOT fbMuestra.Q) ,PT:=T#100MS);
IF fbMuestra.Q AND PV>0 THEN
Volumen:=Volumen+(0.1*PV);
END_IF
IF Reset THEN
	Volumen:=0.0;
	Reset:=0;
END_IF

END_FUNCTION_BLOCK

// ---- POUs/Control Equipos/ControlValv_ioLink.TcPOU
FUNCTION_BLOCK ControlValv_ioLink
VAR_INPUT
	Comando:BOOL;
	Status_1:BYTE;
	Teste:BOOL:=FALSE;
	Inverter:BOOL;
	PosicaoIN:INT;		//Posição da válvula. Valor vindo do IOLink
END_VAR

VAR_OUTPUT
	Estado:INT;
	Falla:BOOL;
	Range:REAL;		//Range de abertura da válvula;
END_VAR

VAR_IN_OUT
	Actuar:BYTE;
END_VAR
VAR
	TemposAcionamento	:ARRAY[1..10] OF DINT;	//Array com os últimos tempos de acionamento
	SwitchCase: INT;
	RTrig: R_TRIG;
	TON_Acionamento: TON;
	iCounter: INT;
	TON_Teste: TON;
	ResetContagem: BOOL;
	PosicaoOUT	:REAL;	//Posição da válvula convertida em %
	IniciarCfg	:BOOL;	//Se a válvula estiver aberta e esse comando for dado, salva o valor de posição como 100%. O mesmo para ela fechada
END_VAR

VAR PERSISTENT
	qntAcionamentos:DINT;	//Quantidade de acionamentos da válvula
	cfgPosicao	:DUT_cfgPosicValvula;		//Configuração de conversão do posicionamento das válvulas
	UltimasPosicoes	:ARRAY[1..2] OF REAL;	//Esse array salva as últimas posições de abertura e fechamento [1] - Abertura, [2] - Fechamento
	
END_VAR

//Acionamento da válvula
Actuar.04 := (Comando AND NOT Inverter) OR (NOT Comando AND Inverter) OR (Teste AND AquecimentoValvulas.Acionar);

TON_Teste(IN:= Actuar.04, PT:= T#465MS);

//Se não estiver em teste, verifica se está aberta, fechada ou em falha
IF NOT Teste THEN
	IF Status_1.0 = 1 THEN	//Válvula aberta
		Estado := 2;
		UltimasPosicoes[1] := PosicaoOUT;	//Salva a posição da válvula no array
	END_IF
	IF Status_1.1 = 1 THEN	//Válvula fechada
		Estado := 1;
		UltimasPosicoes[2] := PosicaoOUT;	//Salva a posição da válvula no array
	END_IF
	IF Status_1.4 = 1 THEN	//Em falha
		Falla := 1;
		Estado := 6;
	END_IF
ELSE
	IF TON_Teste.Q THEN
		Estado := 2;
	ELSE
		Estado := 1;
	END_IF
END_IF

//A lógica abaixo foi feita para calcular o tempo de acionamento da válvula
//Detecta a borda de subida do comando de acionamento
RTrig(CLK:= Actuar.04, Q=> );


//Temporizador do acionamento
TON_Acionamento(IN:= , PT:= T#1M, Q=> , ET=> );

//Se a borda for detectada, inicia a máquina de estados
IF RTRIG.Q THEN
	SwitchCase := 1;
	TON_Acionamento.IN := TRUE;
	//Incrementa os acionamentos
	qntAcionamentos := qntAcionamentos + 1;
END_IF

//Reset da contagem de acionamentos
IF ResetContagem THEN
	qntAcionamentos := 0;
	ResetContagem := FALSE;
END_IF

//Temporizador do acionamento
TON_Acionamento(IN:= , PT:= , Q=> , ET=> );

//Cancela o cálculo se a válvula entrar em falha
IF Falla THEN
	SwitchCase := 0;
END_IF

CASE SwitchCase OF
	1:	IF Estado = 2 THEN
			TemposAcionamento[10] := TIME_TO_DINT(TON_Acionamento.ET);
			SwitchCase := 2;
		END_IF
		
	2:	FOR iCounter := 1 TO 9 BY 1 DO 
			TemposAcionamento[iCounter] := TemposAcionamento[iCounter + 1];
		END_FOR
		TON_Acionamento.IN := FALSE;
		SwitchCase := 0;
END_CASE

//Se a válvula estiver aberta e esse comando for dado, salva o valor de posição como 100%. O mesmo para ela fechada
IF IniciarCfg THEN
	IF Estado = 2 THEN
		cfgPosicao.Aberta := PosicaoIN;
	ELSIF Estado = 1 THEN
		cfgPosicao.Fechada := PosicaoIN;
	END_IF;
	IniciarCfg := FALSE;
END_IF

PosicaoOUT := SEL((cfgPosicao.Aberta - cfgPosicao.Fechada) <> 0,0,(100/(TO_REAL(cfgPosicao.Aberta - cfgPosicao.Fechada))) * (PosicaoIN - cfgPosicao.Fechada));
Range := UltimasPosicoes[1] - UltimasPosicoes[2];		//Calcula o range de abertura da válvula

END_FUNCTION_BLOCK

// ---- POUs/Elementos/Calculo_caudal.TcPOU
FUNCTION_BLOCK Calculo_caudal
VAR_INPUT
	Dosis			:REAL;//ml cada 100Kg
	TiempoInyeccion	:REAL;//segundos
	Peso			:REAL;//en Kg
END_VAR
VAR_OUTPUT
	SetCaudal	:REAL;//ml/s
	Volumen	:REAL;//ml
END_VAR
VAR
END_VAR

Volumen:=Dosis*Peso/100;
IF TiempoInyeccion=0 THEN
	TiempoInyeccion:=1;
END_IF
SetCaudal:=Volumen/TiempoInyeccion;

END_FUNCTION_BLOCK

// ---- POUs/Elementos/CorrecionCaudalxOffset.TcPOU
FUNCTION_BLOCK CorrecionCaudalxOffset
VAR_INPUT
	Caudalimetro_inf	:REAL;
	Caudalimetro_sup	:REAL;	
	Inyeccion			:BOOL;
	Offset				:REAL;
END_VAR
VAR_OUTPUT
	PV					:REAL;
END_VAR
VAR
END_VAR

IF Not Inyeccion THEN
	PV:=Caudalimetro_sup*(Offset+1);
ELSE
	PV:=Caudalimetro_inf*(Offset+1);
END_IF

END_FUNCTION_BLOCK

// ---- POUs/Elementos/FB_PID.TcPOU
FUNCTION_BLOCK FB_PID
VAR_INPUT
	/// Set Point 
	Sp: REAL;
	/// Variable de proceso 
	Pv: REAL;
	/// constante proporcional 
	Kp: REAL := 12;
	/// Tiempo integrativo 
	Ti: REAL := 180;
	/// Tiempo derivativo 
	Td: REAL := 1;
	/// delta de tiempo 
	_dt: REAL := 0.05;
	/// valor minimo de salida 
	_minOut: REAL;
	/// valor máximo de salida 
	_maxOut: REAL;
	/// =1 modo Automatico 
	Auto: BOOL;
	/// reset 
	Reset: BOOL;
	bandaMuerta: REAL;
	PID_Inverso: BOOL;
END_VAR
VAR
	/// error SP-PV
	error: REAL;
	/// diferencial de error para calculo derivativo 
	pre_error: REAL;
	/// proporcional 
	Pout: REAL;
	/// integral
	Iout: REAL;
	/// derivativo 
	Dout: REAL;
	Sp_anterior: REAL;
	Auto_anterior: BOOL;
	Kp_anterior: REAL;
	bandaMuerta_Anterior: REAL;
	bandaMuerta_Sup: REAL;
	Out_anterior:REAL;
	TON_Teste: TON;
	AuxOut: LREAL;
	TestePID: FB_BasicPID;
END_VAR
VAR_IN_OUT
	/// forzar salida manual 
	OutMan: REAL;
END_VAR
VAR_OUTPUT
	/// Salida del lazo 
	Out: REAL;
	///Se llegó al valor del SP
	Sp_Alcanzado: BOOL;
END_VAR

IF (Auto) THEN
	//=== AUTOMATICO ===
	IF PID_Inverso THEN
		error := Pv - Sp;
	ELSE
		error := Sp - Pv;
	END_IF
	
	(* Banda Muerta *)
	IF ( ABS(error) < bandaMuerta ) THEN
		error := 0;
		Sp_Alcanzado:=TRUE;
	ELSE
		Sp_Alcanzado:=FALSE;
	END_IF
	
	(* Termino PROPORCIONAL *)
	Pout := Kp * error;
	
	(* Termino INTEGRAL *)
	IF ( Ti > 0) THEN
		IF ( (Sp_anterior <> Sp) OR (Auto_anterior <> Auto) OR (Kp_anterior <> Kp)) THEN
			(* 
			Parto desde el Iout anterior para evitar el salto y en el proximo scan cambia la pendiente 
			ya sea por el cambio de Sp(nuevo error) o por cambio de parametro Ti.
			*)
			Iout := 0;
		ELSE
			Iout := Iout +( Kp / Ti ) * error * _dt;
		END_IF
	ELSE
		Iout := 0.0;
	END_IF
	 
	(* termino DERIVATIVO *)	
	IF ( _dt > 0.0 AND Td > 0.0) THEN
		IF (Sp = Sp_anterior) THEN
			Dout := Dout + Kp * (error - pre_error);
		END_IF
		Dout := Dout * ( 1 - (_dt / Td ) );

		IF ( ABS(Dout) < (_maxOut / 1000.0)) THEN
			Dout := 0;
		END_IF
	ELSE
		Dout := 0;
	END_IF
	
	(* Salida Lazo de control *)
	//Out := Pout + Out_anterior + Iout + Dout;
	pre_error := error;
END_IF

//Temporizador de teste
	TON_Teste(IN:=Auto, PT:=T#1S);
	
	IF TON_Teste.Q THEN
		Out := SEL(Pout + Out_anterior + Iout + Dout > 0, 0, Pout + Out_anterior + Iout + Dout);
	END_IF
	

// Modo Manual
IF NOT(Auto) THEN
	Out :=  OutMan;
	Sp_Alcanzado:=FALSE;
END_IF

IF ( Pout > _maxOut ) THEN
	Pout := _maxOut;
ELSIF ( Pout < _minOut ) THEN
	Pout := _minOut;
END_IF

(* Restriccion MIN - MAX *)
IF ( Out > _maxOut ) THEN
	Iout := _maxOut;
	Out := _maxOut;
(*ELSIF ( Out < _minOut ) THEN
	Iout := _minOut;
	Out := _minOut;*)
END_IF	

Out_anterior:=Out;	
Auto_anterior := Auto;
Sp_anterior := Sp;
Kp_anterior := Kp;
OutMan := Out;

END_FUNCTION_BLOCK

// ---- POUs/Testes Thiago/Lavagem.TcPOU
FUNCTION_BLOCK Lavagem
VAR_INPUT
	AtivaBloco	:BOOL;	//É acionado quando a linha selecionada é igual a linha definida no programa
	Linha		:INT;	//Linha que o bloco está instanciado
	Status_V1	:INT; //Status da válvula V1
	Status_V2	:INT; //Status da válvula V2
	Status_V3	:INT; //Status da válvula V3
	Status_V4	:INT; //Status da válvula V4
	Status_ValvAguaLimpa:INT; //Status da válvula de água limpa
	Status_ValvAguaResid:INT; //Status da válvula de água residual
	AlarmeBomba	:BOOL; //Alarme da bomba de dosagem
	
	FT_CA	:REAL; //Leitura da vazão após a bomba
	FT_TR	:REAL; //Leitura da vazão antes do tambor
	
END_VAR
VAR_OUTPUT
	Status:INT; //1: Erro nas válvulas, 2: Erro na bomba, 3: Pronto para lavar, 4: Lavando
	Abre_V1:BOOL; //Abre válvula V1
	Abre_V2:BOOL; //Abre válvula V2
	Abre_V3:BOOL; //Abre válvula V3
	Abre_V4:BOOL; //Abre válvula V4
	AguaLimpa:BOOL; //Abre válvula de água limpa
	AguaResid:BOOL; //Abre válvula de água residual
	LigaBombaCW:BOOL; // Aciona bomba em sentido normal
	LigaBombaCCW:BOOL; //Aciona a bomba em sentido contrário
	stStatus:STRING;
	Lavando:BOOL;
	UltimaLav		:LINT;
END_VAR
VAR
	ParaLavagem:BOOL; //Comando para parar a lavagem
	IniciaLavagem:BOOL; //Comando para iniciar a lavagem
	SwitchCase :INT:=0; //Variável para iteração no case
	TON1_Lavagem: TON; //Temporizador 1
	TON2_Lavagem: TON; //Temporizador 2
	TON3_Lavagem: TON; //Temporizador 3
	TON4_Lavagem: TON; //Temporizador 4
	TON5_Lavagem: TON; //Temporizador 5
	TON6_Lavagem: TON;	//Temporizador 6
	TONR6_Lavagem	:TONR;	//Temporizador retentivo
	QntLavResid: INT := 0; //Quantidade de lavagens feitas com água residual
	QntLavLimpa: INT := 0; //Quantidade de lavagens feitas com água limpa
	TempoTotal:REAL;		//Cálculo do tempo total da lavagem
	TempoAtual:REAL;		//Tempo decorrido da lavagem atual
	PorcentLavagem	:REAL;	//percentual de conclusão da lavagem
END_VAR
VAR PERSISTENT
	Config:DUT_ConfigLavagem; //Variável com as configurações de lavagem
	UltimaLavagem	:UDINT;	//Data e hora da última lavagem - //Estão como UDINT para a correta conversão na IHM
	IntervLavagem	:UDINT;	//Intervalo entre lavagens (h)
END_VAR

UltimaLav := UltimaLavagem;

//Se o alarme lavagem subir, o próximo alarme da mesma linha será no próximo intervalo
(*
IF IntervaloLavCalibr.AlarmeLavagem AND IntervaloLavCalibr.LinhaLavagem = Linha THEN
	UltimaLavagem := DT_TO_UDINT(Main.HoraAtual);
END_IF*)

//Status da lavagem
IF Status_V2 = 6 OR Status_V3 = 6 OR Status_V4 = 6 OR Status_ValvAguaLimpa = 6 OR Status_ValvAguaResid = 6 OR TON5_Lavagem.Q THEN
	Status := 1; // Problema nas válvulas
	stStatus := 'FALHA NO POSICIONAMENTO DAS VÁLVULAS';
ELSIF AlarmeBomba THEN
	Status := 2; //Problema na bomba
	stStatus := 'PROBLEMA NA BOMBA';
ELSIF (Config.LavAguaLimpa <= 0 AND Config.LavAguaUsada <= 0) OR (Config.TempoDeCiclo) <= 0 THEN
	Status := 7; //Problema nas configurações do ciclo
	stStatus := 'PROBLEMA NAS CONFIGURAÇÕES DO CICLO';
ELSIF SwitchCase = 0 THEN
	Status := 3; //Pronto para iniciar lavagem
	stStatus := 'PRONTO PARA INICIAR LAVAGEM';
ELSIF SwitchCase > 0 AND SwitchCase < 30 THEN
	Status := 4; //Lavagem com água residual
	stStatus := 'LAVANDO COM ÁGUA RESIDUAL';
ELSIF SwitchCase >= 30 AND SwitchCase < 42 THEN
	Status := 5; //Lavagem com água limpa
	stStatus := 'LAVANDO COM ÁGUA LIMPA';
ELSE
	Status := 6; //Finalizando lavagem
	stStatus := 'FINALIZANDO LAVAGEM';
END_IF;
/// Colocar o que falta para iniciar a lavagem

//Cálculo do tempo total de lavagem
TempoTotal := DINT_TO_REAL(2 * (Config.TempoDeCiclo + 1) * ( Config.LavAguaLimpa + Config.LavAguaUsada)) + TIME_TO_REAL(TON4_Lavagem.PT/1000);
TempoAtual := (TIME_TO_REAL(TONR6_Lavagem.ACC)/1000);
IF TempoTotal <> 0 THEN
	PorcentLavagem := ((TempoAtual)/(TempoTotal)) * 100;
END_IF


// Instância dos timers
TON1_Lavagem(IN:= LigaBombaCW, PT:= DINT_TO_TIME(Config.TempoDeCiclo)*1000, Q=> , ET=> ); 
TON2_Lavagem(IN:= LigaBombaCCW, PT:= DINT_TO_TIME(Config.TempoDeCiclo)*1000, Q=> , ET=> );
TON3_Lavagem(IN:= , PT:= T#1S, Q=> , ET=> ); //Tempo entre a reversão das bombas
TON4_Lavagem(IN:= , PT:= T#5S, Q=> , ET=> ); //Timer de finalização da lavagem
TON5_Lavagem(IN:= , PT:= T#10S, Q=> , ET=> );	//Temporizador para esperar as válvulas posicionarem
TON6_Lavagem(IN:= (SwitchCase >= 10 AND SwitchCase < 42), PT:= REAL_TO_TIME(TempoTotal * 1000), Q=> , ET=> );	//Tempo total da lavagem
TONR6_Lavagem(
	EN:= (SwitchCase >= 10 AND SwitchCase <= 42) AND NOT TON5_Lavagem.IN, 
	PRE:= REAL_TO_TIME(TempoTotal * 1000), 
	RES:= TONR6_Lavagem.DN OR SwitchCase = 0, 
	DN=> , 
	ACC=> , 
	TT=> );


//Verifica condições para iniciar lavagem
IF Status = 3 AND IniciaLavagem AND NOT ParaLavagem AND AtivaBloco THEN
	IniciaLavagem := FALSE;
	IF Config.LavAguaUsada = 0 THEN
		SwitchCase := 30;
	ELSE
		SwitchCase := 10;
	END_IF
END_IF

//Para a lavagem
IF (ParaLavagem AND AtivaBloco) THEN //Deve ter o AtivaBLoco para que só a linha selecionada pare de lavar
	SwitchCase := 0;
	ParaLavagem := FALSE;
	HMI.PararLavagem := FALSE;
	TON5_Lavagem.IN := FALSE;	//Reseta falha no posicionamento das válvulas
END_IF

//Se a linha estiver sendo lavada e o bloco é desativado, a bomba deve retornar o material antes de parar
IF Lavando AND NOT AtivaBloco AND SwitchCase < 31 AND SwitchCase <> 0 THEN
	IniciaLavagem := False;
	SwitchCase := 31;
END_IF

CASE SwitchCase OF
	
	0:	//Sistema parado
		AguaLimpa := FALSE;
		AguaResid := FALSE;
		LigaBombaCW := FALSE;
		LigaBombaCCW := FALSE;
		QntLavResid := 0;
		QntLavLimpa := 0;
		Lavando := FALSE;
		IniciaLavagem := FALSE;
		
	10: //Inicia a lavagem com água residual
		Abre_V1 := TRUE;
		Abre_V2 := TRUE;
		Abre_V3 := FALSE;
		AguaLimpa := FALSE;
		AguaResid := TRUE; 
		Lavando := TRUE;
		
		//Verifica se todas as válvulas abriram
		IF Status_V1 = 2 AND Status_V2 = 2 AND Status_V3 = 1 AND Status_ValvAguaResid = 2 THEN
			LigaBombaCW := TRUE;
			LigaBombaCCW :=  FALSE;
			TON5_Lavagem.IN := FALSE;
		ELSE
			stStatus := 'AGUARDANDO VÁLVULAS POSICIONAREM';
			Status := 8;
			TON5_Lavagem.IN := TRUE;
			IF TON5_Lavagem.Q THEN
				SwitchCase := 0;
			END_IF
		END_IF
		
		IF TON1_Lavagem.Q THEN
			SwitchCase := 11;
		END_IF
		
	11: TON3_Lavagem.IN := TRUE;		//Bloco de espera para a reversão do motor
		LigaBombaCW := FALSE;
		LigaBombaCCW :=  FALSE;
		IF TON3_Lavagem.Q THEN
			SwitchCase := 20;
			TON3_Lavagem.IN := FALSE;
		END_IF
		
	20: //Giro reverso
		LigaBombaCW := FALSE;
		LigaBombaCCW :=  TRUE;
		
		IF TON2_Lavagem.Q THEN
			QntLavResid := QntLavResid + 1;
			IF QntLavResid < Config.LavAguaUsada THEN
				SwitchCase := 21;
			ELSE
				SwitchCase := 22;
			END_IF
		END_IF
		
	21: TON3_Lavagem.IN	:= TRUE;		//Bloco de espera para a reversão do motor
		LigaBombaCW		:= FALSE;
		LigaBombaCCW 	:=  FALSE;
		IF TON3_Lavagem.Q THEN
			SwitchCase := 10;
			TON3_Lavagem.IN := FALSE;
		END_IF
		
	22: TON3_Lavagem.IN := TRUE;		//Bloco de espera para a reversão do motor
		LigaBombaCW 	:= FALSE;
		LigaBombaCCW 	:=  FALSE;
		IF TON3_Lavagem.Q THEN
			SwitchCase := 30;
			TON3_Lavagem.IN := FALSE;
		END_IF
		
	30: Abre_V1 := TRUE;
		Abre_V2 := FALSE;
		Abre_V3 := FALSE;
		AguaLimpa := TRUE;
		AguaResid := FALSE;
		Lavando := TRUE;
		
		IF Status_V1 = 2 AND Status_V2 = 1 AND Status_V3 = 1 AND Status_ValvAguaLimpa = 2 THEN
			LigaBombaCW := TRUE;
			LigaBombaCCW :=  FALSE;
			TON5_Lavagem.IN := FALSE;
		ELSE
			stStatus := 'AGUARDANDO POSICIONAMENTO DAS VÁLVULAS';
			Status := 8;
			TON5_Lavagem.IN := TRUE;
			IF TON5_Lavagem.Q THEN
				SwitchCase := 0;
			END_IF
		END_IF
		
		IF TON1_Lavagem.Q THEN
			SwitchCase := 31;
			Abre_V2 := TRUE;
			Abre_V3 := FALSE;
			Abre_V4 := TRUE;
			AguaLimpa := FALSE;
			AguaResid := TRUE;
		END_IF
	
	31: TON3_Lavagem.IN := TRUE;		//Bloco de espera para a reversão do motor
		LigaBombaCW := FALSE;
		LigaBombaCCW :=  FALSE;
		IF TON3_Lavagem.Q THEN
			SwitchCase := 40;
			TON3_Lavagem.IN := FALSE;
		END_IF
		
	40: LigaBombaCW := FALSE;	//A água limpa, deve retornar para o recipiente de água residual
		LigaBombaCCW :=  TRUE;
		
		
		IF TON2_Lavagem.Q THEN
			QntLavLimpa := QntLavLimpa + 1;
			IF (QntLavLimpa < Config.LavAguaLimpa) AND AtivaBloco THEN
				SwitchCase := 41;
				Abre_V1 := TRUE;
				Abre_V2 := FALSE;
				Abre_V3 := FALSE;
				AguaLimpa := TRUE;
				AguaResid := FALSE;
			ELSE
				SwitchCase := 42;
			END_IF
			IF NOT AtivaBloco THEN
				SwitchCase := 42;
			END_IF
		END_IF
		
	41: TON3_Lavagem.IN := TRUE;		//Bloco de espera para a reversão do motor
		LigaBombaCW := FALSE;
		LigaBombaCCW :=  FALSE;
		IF TON3_Lavagem.Q THEN
			SwitchCase := 30;
			TON3_Lavagem.IN := FALSE;
		END_IF
		
	42: TON4_Lavagem.IN := TRUE; // Finalização da lavagem
		UltimaLavagem := DT_TO_UDINT(MAIN.HoraAtual);	//Verifica a hora que a ultima lavagem foi feita
		Liquidos.UltimoAlrLavagem[Linha] := DT_TO_LINT(MAIN.HoraAtual);
		Abre_V1 := FALSE;
		Abre_V2 := FALSE;
		Abre_V3 := FALSE;
		Abre_V4 := FALSE;
		IF TON4_Lavagem.Q THEN
			SwitchCase := 0;
			TON4_Lavagem.IN := FALSE;
			IniciaLavagem := FALSE;
		END_IF
		
	
END_CASE

END_FUNCTION_BLOCK

// ---- POUs/Testes Thiago/Filtro2.TcPOU
FUNCTION_BLOCK Filtro2
VAR_INPUT
	Input:REAL;	//Entrada do sensor
	Tempo:DINT := 500;	//Tempo de amostragem
END_VAR
VAR
	Amostras:ARRAY[1..50] OF REAL;
	TON_Amostras:TON;
	i		:INT;	//Variável de iteração do FOR
	Soma 	:REAL;	//Somatório dos valores do array
	Teste: INT;
END_VAR
VAR_OUTPUT
	Output:REAL;
END_VAR

TON_Amostras(IN := NOT TON_Amostras.Q, PT:=DINT_TO_TIME(Tempo));

IF TON_Amostras.Q THEN
	//Faz o shift do array
	FOR i := 1 TO 49 DO
		Amostras[i] := Amostras[i + 1];
	END_FOR
	
	//Insere a leitura do sensor na última posição
	Amostras[50] := Input;
	
	//Soma os valores do array
	Soma := 0;
	FOR i := 1 TO 50 DO
		Soma := Soma + Amostras[i];
	END_FOR
	
	Output := Soma / 50;
END_IF

END_FUNCTION_BLOCK

// ---- POUs/Testes Thiago/LiqNaReceita.TcPOU
PROGRAM LiqNaReceita
VAR
	iCounter: INT;
END_VAR

//Esse bloco verifica quais liquidos que estão sendo usados na receita, para que não seja possível iniciar a limpeza neles
FOR iCounter := 1 TO 12 DO
		Liquidos.LiqNaReceita[iCounter] := Receta_Activa.SetCircuitosLiq[iCounter].Paso <> 0;
END_FOR

END_PROGRAM

// ---- POUs/Lavado/Valvulas_Lavado.TcPOU
PROGRAM Valvulas_Lavado
VAR
	ControlValv_ioLink_V6: ControlValv_ioLink;
	Falla_Lav_V6: BOOL;
	ControlValv_ioLink_V5: ControlValv_ioLink;
	Falla_Lav_V5: BOOL;
END_VAR
VAR // added by the converter: edge detectors and wires of the graphical bodies
    _w1, _w2 : BOOL;
END_VAR

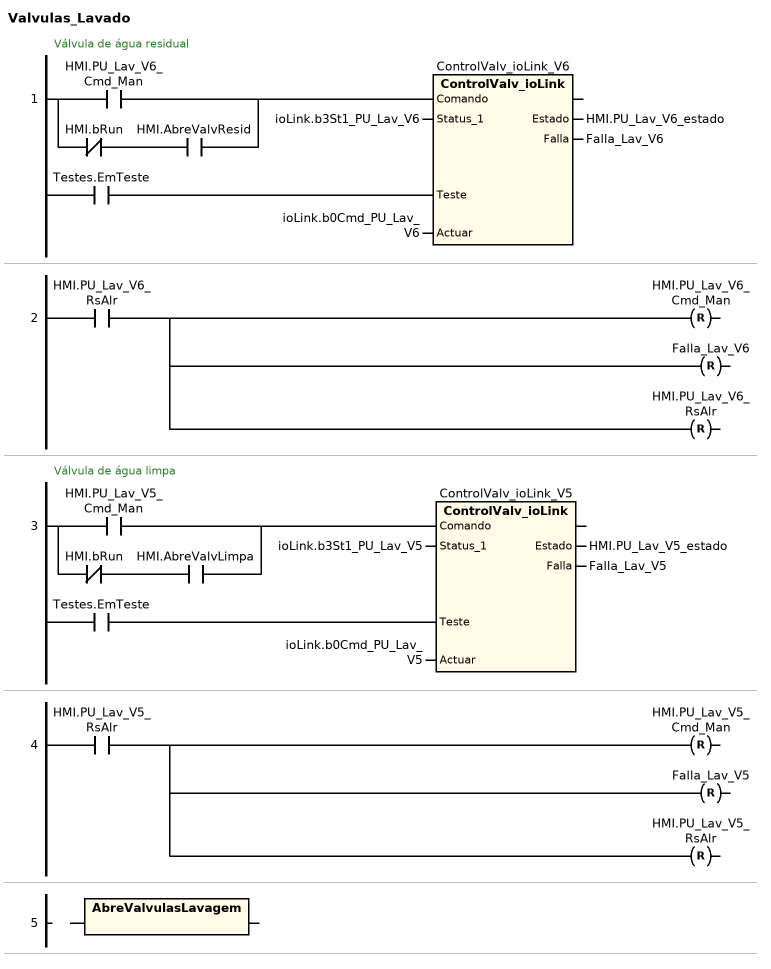
// NETWORK 1
// Válvula de água residual
ControlValv_ioLink_V6(
    Comando := HMI.PU_Lav_V6_Cmd_Man OR NOT HMI.bRun AND HMI.AbreValvResid,
    Status_1 := ioLink.b3St1_PU_Lav_V6,
    Teste := Testes.EmTeste,
    Actuar := ioLink.b0Cmd_PU_Lav_V6,
    Estado => HMI.PU_Lav_V6_estado,
    Falla => Falla_Lav_V6); // ControlValv_ioLink

// NETWORK 2
_w1 := HMI.PU_Lav_V6_RsAlr;
HMI.PU_Lav_V6_Cmd_Man R= _w1;
Falla_Lav_V6 R= _w1;
HMI.PU_Lav_V6_RsAlr R= _w1;

// NETWORK 3
// Válvula de água limpa
ControlValv_ioLink_V5(
    Comando := HMI.PU_Lav_V5_Cmd_Man OR NOT HMI.bRun AND HMI.AbreValvLimpa,
    Status_1 := ioLink.b3St1_PU_Lav_V5,
    Teste := Testes.EmTeste,
    Actuar := ioLink.b0Cmd_PU_Lav_V5,
    Estado => HMI.PU_Lav_V5_estado,
    Falla => Falla_Lav_V5); // ControlValv_ioLink

// NETWORK 4
_w2 := HMI.PU_Lav_V5_RsAlr;
HMI.PU_Lav_V5_Cmd_Man R= _w2;
Falla_Lav_V5 R= _w2;
HMI.PU_Lav_V5_RsAlr R= _w2;

// NETWORK 5
AbreValvulasLavagem();

END_PROGRAM

// ---- POUs/Lavado/AbreValvulasLavagem.TcPOU
PROGRAM AbreValvulasLavagem
VAR
END_VAR

HMI.AbreValvLimpa :=	   Circuito_L1.Lavagem_Circuito01.AguaLimpa 
						OR Circuito_L2.Lavagem_Circuito02.AguaLimpa
						OR Circuito_L3.Lavagem_Circuito03.AguaLimpa
						OR Circuito_L4.Lavagem_Circuito04.AguaLimpa //Colocar aqui todos os contatos que abre a válvula pertinente
						OR Circuito_L5.Lavagem_Circuito05.AguaLimpa
						OR Circuito_L6.Lavagem_Circuito06.AguaLimpa
						OR Circuito_L7.Lavagem_Circuito07.AguaLimpa
						OR Circuito_L8.Lavagem_Circuito08.AguaLimpa
						OR Circuito_L9.Lavagem_Circuito9.AguaLimpa
						OR Circuito_L10.Lavagem_Circuito10.AguaLimpa
						OR Circuito_L11.Lavagem_Circuito11.AguaLimpa
						OR Circuito_L12.Lavagem_Circuito12.AguaLimpa;
						
HMI.AbreValvResid :=       Circuito_L1.Lavagem_Circuito01.AguaResid
						OR Circuito_L2.Lavagem_Circuito02.AguaResid
						OR Circuito_L3.Lavagem_Circuito03.AguaResid
						OR Circuito_L4.Lavagem_Circuito04.AguaResid
						OR Circuito_L5.Lavagem_Circuito05.AguaResid
						OR Circuito_L6.Lavagem_Circuito06.AguaResid
						OR Circuito_L7.Lavagem_Circuito07.AguaResid
						OR Circuito_L8.Lavagem_Circuito08.AguaResid
						OR Circuito_L9.Lavagem_Circuito9.AguaResid
						OR Circuito_L10.Lavagem_Circuito10.AguaResid
						OR Circuito_L11.Lavagem_Circuito11.AguaResid
						OR Circuito_L12.Lavagem_Circuito12.AguaResid;

END_PROGRAM

// ---- POUs/Puesto_Calibracion_1/Circuito_L2.TcPOU
PROGRAM Circuito_L2
VAR_INPUT
	Modo_Calibrar_L2: BOOL;
END_VAR

VAR
		fbBomba_L2 :Equipo_Motor_ATV320;
		ControlValv_ioLink_V1:ControlValv_ioLink;
		ControlValv_ioLink_V2: ControlValv_ioLink;
		ControlValv_ioLink_V3: ControlValv_ioLink;
		ControlValv_ioLink_V4: ControlValv_ioLink;
		Falla_L2_V1:BOOL;
		Falla_L2_V2:BOOL;
		Falla_L2_V3:BOOL;
		Falla_L2_V4:BOOL;
	Balanza_PU1_WT2: Balanza;
		dHS:DINT;
		TOF_calibradoIBC: TOF;
		TDemoraInyectar: TON;
		SetDemoraInyeccion: REAL;	
	Volumen_L2: REAL;
	AuxVol: REAL;
	Total: REAL;
	auxIniCal: BOOL;
	Calculo_caudal_L2: Calculo_caudal;
	PID_L2_SP: REAL;
	PID_L2_PV: REAL;
	CorrecionCaudalxOffset_L2: CorrecionCaudalxOffset;
	tInyeccion: TON;
	PID_L2_manual: REAL;
	PID_L2: FB_PID;
	PID_L2_Kp: REAL := 0.1;
	PID_L2_Ti: REAL := 100;
	PID_L2_auto: BOOL;
	PID_L2_reset: BOOL;
	PID_L2_bMuerta: REAL := 5;
	Tiempo_seg_to_TIME_DemoraInyec: Tiempo_seg_to_TIME;
	AuxTDemoraInyec: TIME;
	Tiempo_TIME_to_seg_InyCal: Tiempo_TIME_to_seg;
	AuxInyCal:TIME;
	ProductoAsociado:STRING;

	Lavagem_Circuito02: Lavagem;
END_VAR
VAR PERSISTENT
	UltimaCalibracao	:UDINT;	//Data e hora da ultima calibração
END_VAR
VAR // added by the converter: edge detectors and wires of the graphical bodies
    _w1, _w2, _w3, _w4, _w5, _w6, _w7, _w8, _w9, _w10, _w11, _w12, _w13 : BOOL;
    _ft1 : F_TRIG;
    _rt1 : R_TRIG;
END_VAR

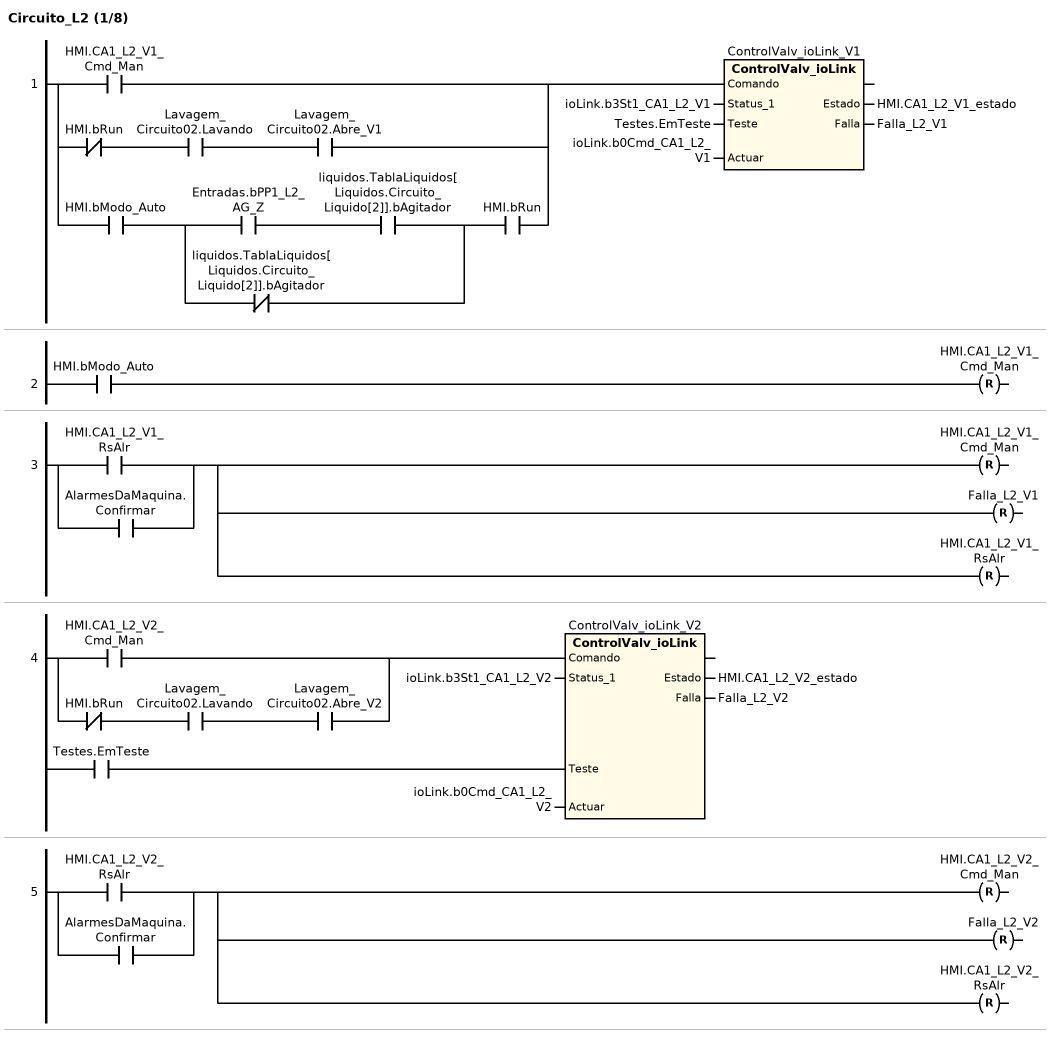
// NETWORK 1
ControlValv_ioLink_V1(
    Comando := HMI.CA1_L2_V1_Cmd_Man OR NOT HMI.bRun AND Lavagem_Circuito02.Lavando AND Lavagem_Circuito02.Abre_V1 OR HMI.bModo_Auto AND (Entradas.bPP1_L2_AG_Z AND (liquidos.TablaLiquidos[Liquidos.Circuito_Liquido[2]].bAgitador) OR NOT (liquidos.TablaLiquidos[Liquidos.Circuito_Liquido[2]].bAgitador)) AND HMI.bRun,
    Status_1 := ioLink.b3St1_CA1_L2_V1,
    Teste := Testes.EmTeste,
    Actuar := ioLink.b0Cmd_CA1_L2_V1,
    Estado => HMI.CA1_L2_V1_estado,
    Falla => Falla_L2_V1); // ControlValv_ioLink

// NETWORK 2
HMI.CA1_L2_V1_Cmd_Man R= HMI.bModo_Auto;

// NETWORK 3
_w1 := HMI.CA1_L2_V1_RsAlr OR AlarmesDaMaquina.Confirmar;
HMI.CA1_L2_V1_Cmd_Man R= _w1;
Falla_L2_V1 R= _w1;
HMI.CA1_L2_V1_RsAlr R= _w1;

// NETWORK 4
ControlValv_ioLink_V2(
    Comando := HMI.CA1_L2_V2_Cmd_Man OR NOT HMI.bRun AND Lavagem_Circuito02.Lavando AND Lavagem_Circuito02.Abre_V2,
    Status_1 := ioLink.b3St1_CA1_L2_V2,
    Teste := Testes.EmTeste,
    Actuar := ioLink.b0Cmd_CA1_L2_V2,
    Estado => HMI.CA1_L2_V2_estado,
    Falla => Falla_L2_V2); // ControlValv_ioLink

// NETWORK 5
_w2 := HMI.CA1_L2_V2_RsAlr OR AlarmesDaMaquina.Confirmar;
HMI.CA1_L2_V2_Cmd_Man R= _w2;
Falla_L2_V2 R= _w2;
HMI.CA1_L2_V2_RsAlr R= _w2;

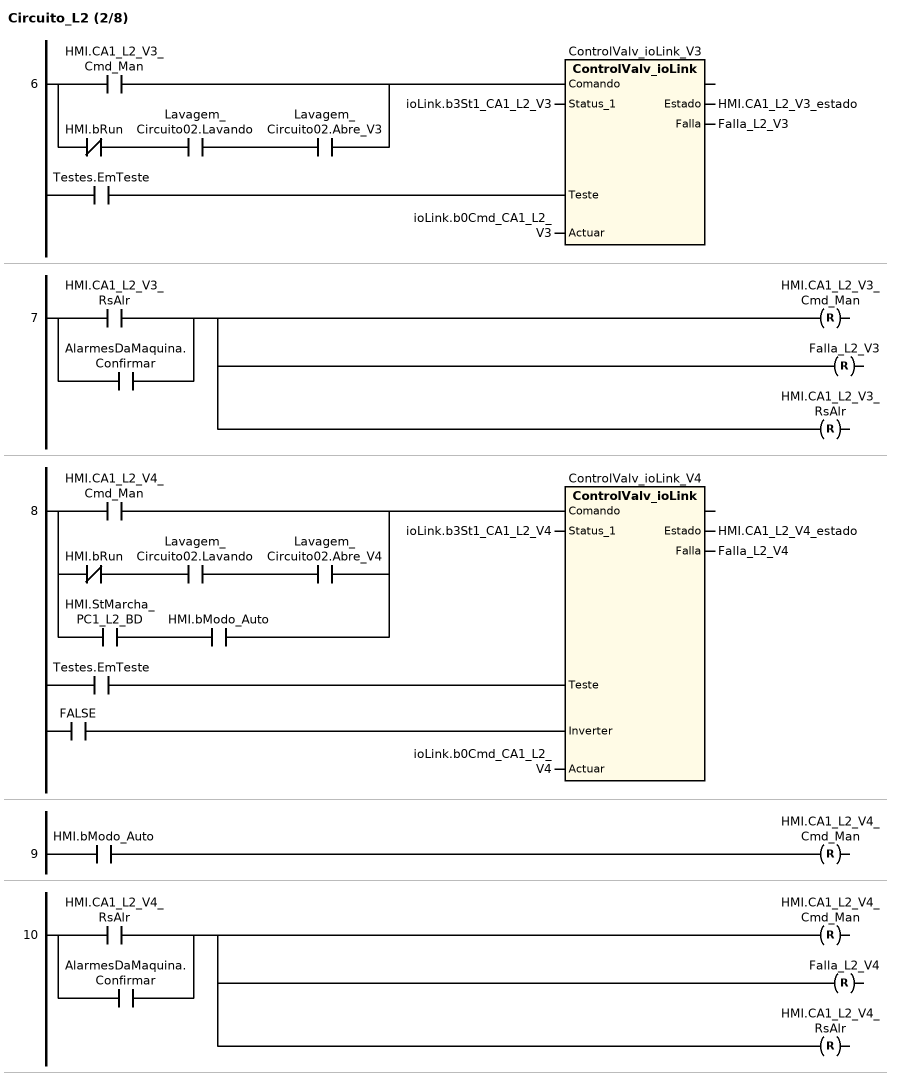
// NETWORK 6
ControlValv_ioLink_V3(
    Comando := HMI.CA1_L2_V3_Cmd_Man OR NOT HMI.bRun AND Lavagem_Circuito02.Lavando AND Lavagem_Circuito02.Abre_V3,
    Status_1 := ioLink.b3St1_CA1_L2_V3,
    Teste := Testes.EmTeste,
    Actuar := ioLink.b0Cmd_CA1_L2_V3,
    Estado => HMI.CA1_L2_V3_estado,
    Falla => Falla_L2_V3); // ControlValv_ioLink

// NETWORK 7
_w3 := HMI.CA1_L2_V3_RsAlr OR AlarmesDaMaquina.Confirmar;
HMI.CA1_L2_V3_Cmd_Man R= _w3;
Falla_L2_V3 R= _w3;
HMI.CA1_L2_V3_RsAlr R= _w3;

// NETWORK 8
ControlValv_ioLink_V4(
    Comando := HMI.CA1_L2_V4_Cmd_Man OR NOT HMI.bRun AND Lavagem_Circuito02.Lavando AND Lavagem_Circuito02.Abre_V4 OR HMI.StMarcha_PC1_L2_BD AND HMI.bModo_Auto,
    Status_1 := ioLink.b3St1_CA1_L2_V4,
    Teste := Testes.EmTeste,
    Inverter := FALSE,
    Actuar := ioLink.b0Cmd_CA1_L2_V4,
    Estado => HMI.CA1_L2_V4_estado,
    Falla => Falla_L2_V4); // ControlValv_ioLink

// NETWORK 9
HMI.CA1_L2_V4_Cmd_Man R= HMI.bModo_Auto;

// NETWORK 10
_w4 := HMI.CA1_L2_V4_RsAlr OR AlarmesDaMaquina.Confirmar;
HMI.CA1_L2_V4_Cmd_Man R= _w4;
Falla_L2_V4 R= _w4;
HMI.CA1_L2_V4_RsAlr R= _w4;

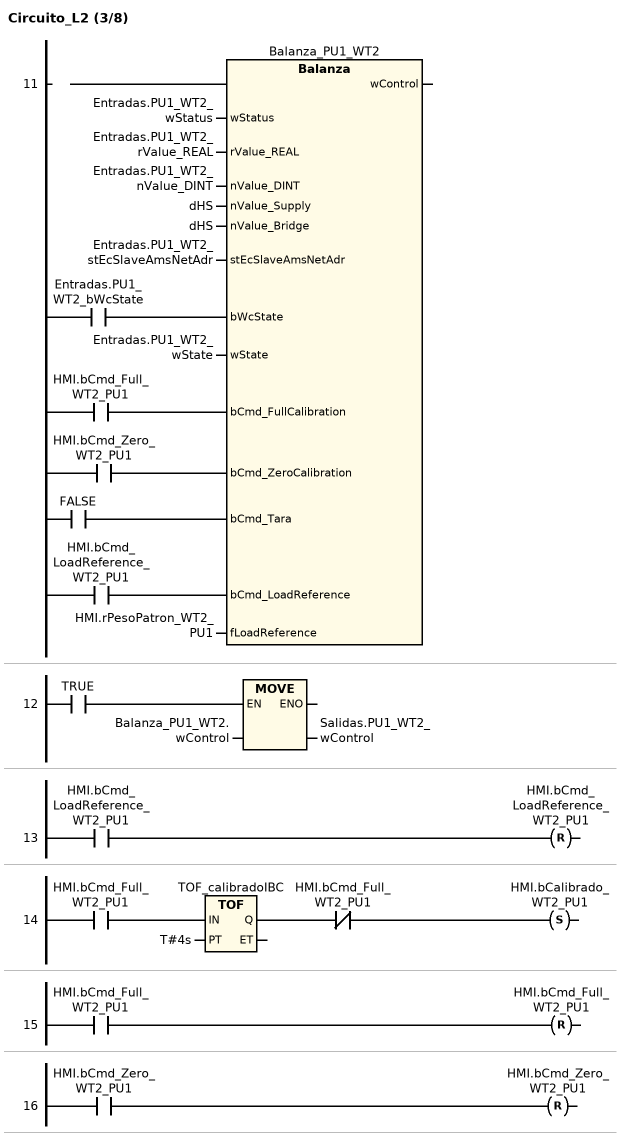
// NETWORK 11
Balanza_PU1_WT2(
    wStatus := Entradas.PU1_WT2_wStatus,
    rValue_REAL := Entradas.PU1_WT2_rValue_REAL,
    nValue_DINT := Entradas.PU1_WT2_nValue_DINT,
    nValue_Supply := dHS,
    nValue_Bridge := dHS,
    stEcSlaveAmsNetAdr := Entradas.PU1_WT2_stEcSlaveAmsNetAdr,
    bWcState := Entradas.PU1_WT2_bWcState,
    wState := Entradas.PU1_WT2_wState,
    bCmd_FullCalibration := HMI.bCmd_Full_WT2_PU1,
    bCmd_ZeroCalibration := HMI.bCmd_Zero_WT2_PU1,
    bCmd_Tara := FALSE,
    bCmd_LoadReference := HMI.bCmd_LoadReference_WT2_PU1,
    fLoadReference := HMI.rPesoPatron_WT2_PU1); // Balanza

// NETWORK 12
Salidas.PU1_WT2_wControl := Balanza_PU1_WT2.wControl;

// NETWORK 13
HMI.bCmd_LoadReference_WT2_PU1 R= HMI.bCmd_LoadReference_WT2_PU1;

// NETWORK 14
TOF_calibradoIBC(IN := HMI.bCmd_Full_WT2_PU1, PT := T#4s); // TOF
HMI.bCalibrado_WT2_PU1 S= TOF_calibradoIBC.Q AND NOT HMI.bCmd_Full_WT2_PU1;

// NETWORK 15
HMI.bCmd_Full_WT2_PU1 R= HMI.bCmd_Full_WT2_PU1;

// NETWORK 16
HMI.bCmd_Zero_WT2_PU1 R= HMI.bCmd_Zero_WT2_PU1;

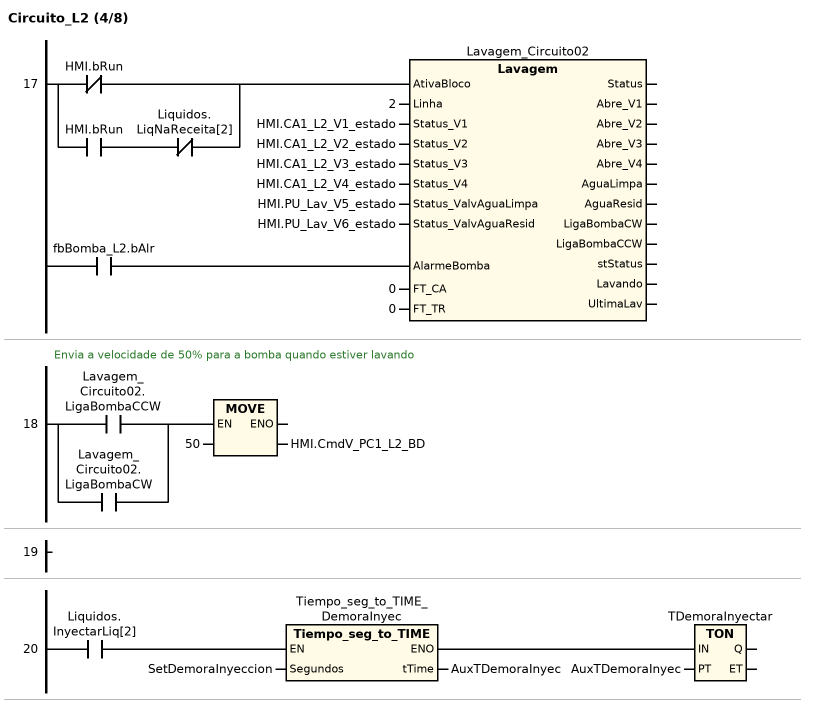
// NETWORK 17
Lavagem_Circuito02(
    AtivaBloco := NOT HMI.bRun OR HMI.bRun AND NOT Liquidos.LiqNaReceita[2],
    Linha := 2,
    Status_V1 := HMI.CA1_L2_V1_estado,
    Status_V2 := HMI.CA1_L2_V2_estado,
    Status_V3 := HMI.CA1_L2_V3_estado,
    Status_V4 := HMI.CA1_L2_V4_estado,
    Status_ValvAguaLimpa := HMI.PU_Lav_V5_estado,
    Status_ValvAguaResid := HMI.PU_Lav_V6_estado,
    AlarmeBomba := fbBomba_L2.bAlr,
    FT_CA := 0,
    FT_TR := 0); // Lavagem

// NETWORK 18
// Envia a velocidade de 50% para a bomba quando estiver lavando
IF Lavagem_Circuito02.LigaBombaCCW OR Lavagem_Circuito02.LigaBombaCW THEN HMI.CmdV_PC1_L2_BD := 50; END_IF

// NETWORK 19

// NETWORK 20
_w5 := Liquidos.InyectarLiq[2];
IF _w5 THEN
    Tiempo_seg_to_TIME_DemoraInyec(Segundos := SetDemoraInyeccion, tTime => AuxTDemoraInyec); // Tiempo_seg_to_TIME
END_IF
TDemoraInyectar(IN := _w5, PT := AuxTDemoraInyec); // TON

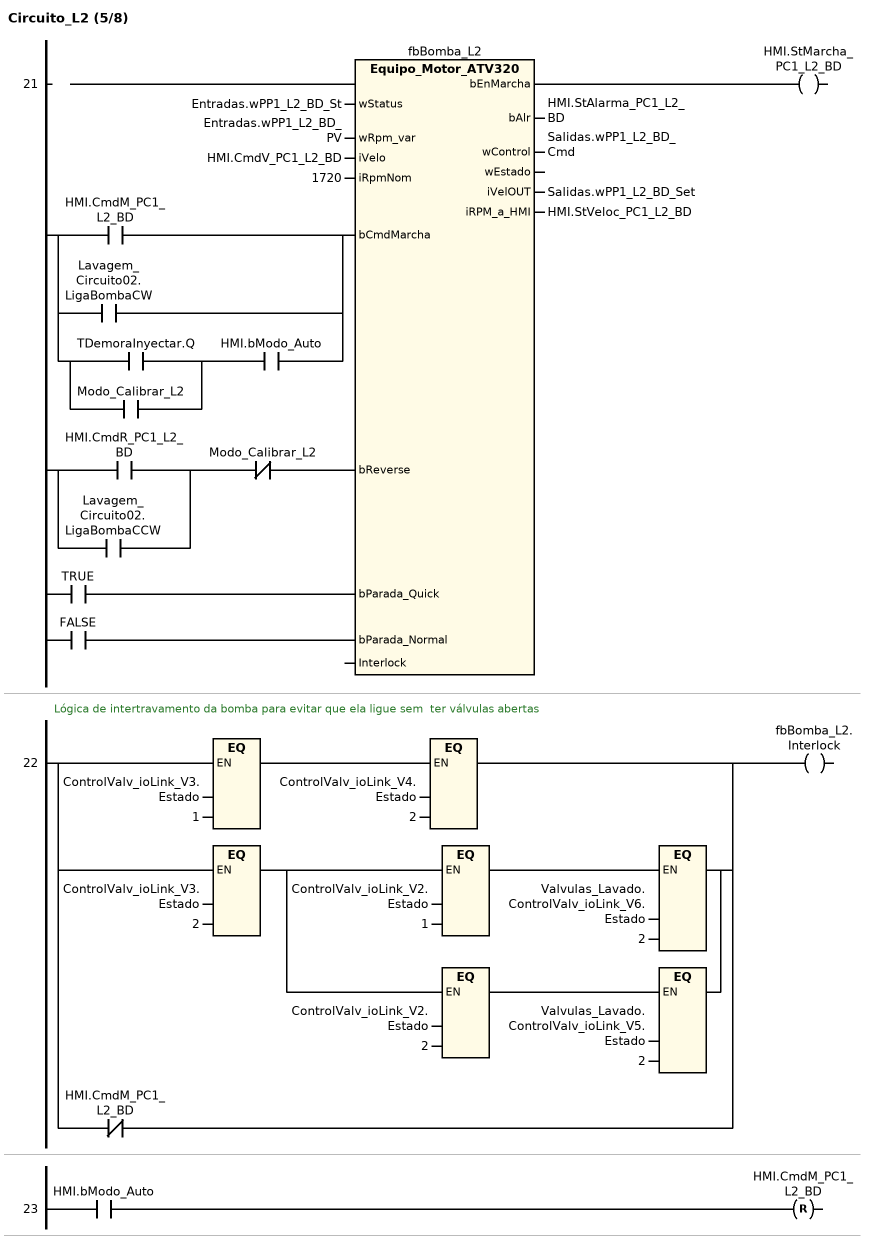
// NETWORK 21
fbBomba_L2(
    wStatus := Entradas.wPP1_L2_BD_St,
    wRpm_var := Entradas.wPP1_L2_BD_PV,
    iVelo := HMI.CmdV_PC1_L2_BD,
    iRpmNom := 1720,
    bCmdMarcha := HMI.CmdM_PC1_L2_BD OR Lavagem_Circuito02.LigaBombaCW OR (TDemoraInyectar.Q OR Modo_Calibrar_L2) AND HMI.bModo_Auto,
    bReverse := (HMI.CmdR_PC1_L2_BD OR Lavagem_Circuito02.LigaBombaCCW) AND NOT Modo_Calibrar_L2,
    bParada_Quick := TRUE,
    bParada_Normal := FALSE,
    bAlr => HMI.StAlarma_PC1_L2_BD,
    wControl => Salidas.wPP1_L2_BD_Cmd,
    iVelOUT => Salidas.wPP1_L2_BD_Set,
    iRPM_a_HMI => HMI.StVeloc_PC1_L2_BD); // Equipo_Motor_ATV320
HMI.StMarcha_PC1_L2_BD := fbBomba_L2.bEnMarcha;

// NETWORK 22
// Lógica de intertravamento da bomba para evitar que ela ligue sem  ter válvulas abertas
_w6 := NOT HMI.CmdM_PC1_L2_BD;
IF NOT _w6 THEN
    _w7 := ControlValv_ioLink_V3.Estado = 2;
    _w6 := ControlValv_ioLink_V3.Estado = 1 AND ControlValv_ioLink_V4.Estado = 2 OR (_w7 AND ControlValv_ioLink_V2.Estado = 1 AND Valvulas_Lavado.ControlValv_ioLink_V6.Estado = 2 OR _w7 AND ControlValv_ioLink_V2.Estado = 2 AND Valvulas_Lavado.ControlValv_ioLink_V5.Estado = 2);
END_IF
fbBomba_L2.Interlock := _w6;

// NETWORK 23
HMI.CmdM_PC1_L2_BD R= HMI.bModo_Auto;

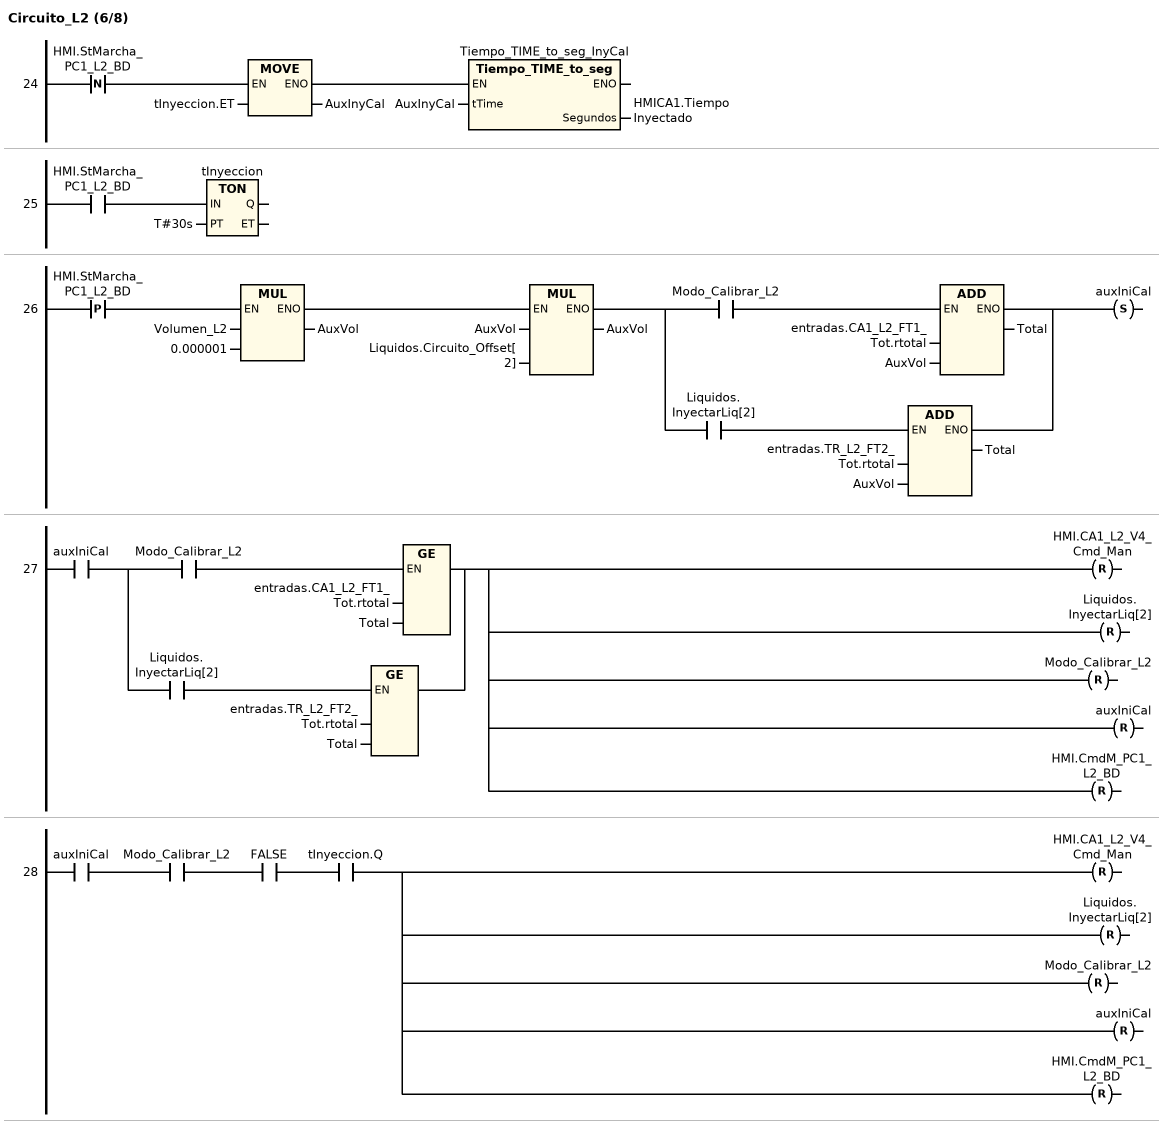
// NETWORK 24
_ft1(CLK := HMI.StMarcha_PC1_L2_BD);
_w8 := _ft1.Q;
IF _w8 THEN AuxInyCal := tInyeccion.ET; END_IF
IF _w8 THEN
    Tiempo_TIME_to_seg_InyCal(tTime := AuxInyCal, Segundos => HMICA1.TiempoInyectado); // Tiempo_TIME_to_seg
END_IF

// NETWORK 25
tInyeccion(IN := HMI.StMarcha_PC1_L2_BD, PT := T#30s); // TON

// NETWORK 26
_rt1(CLK := HMI.StMarcha_PC1_L2_BD);
_w9 := _rt1.Q;
IF _w9 THEN AuxVol := Volumen_L2 * 0.000001; END_IF
IF _w9 THEN AuxVol := AuxVol * Liquidos.Circuito_Offset[2]; END_IF
IF _w9 AND Modo_Calibrar_L2 THEN Total := entradas.CA1_L2_FT1_Tot.rtotal + AuxVol; END_IF
IF _w9 AND Liquidos.InyectarLiq[2] THEN Total := entradas.TR_L2_FT2_Tot.rtotal + AuxVol; END_IF
auxIniCal S= _w9 AND Modo_Calibrar_L2 OR _w9 AND Liquidos.InyectarLiq[2];

// NETWORK 27
_w10 := auxIniCal AND Modo_Calibrar_L2 AND entradas.CA1_L2_FT1_Tot.rtotal >= Total OR auxIniCal AND Liquidos.InyectarLiq[2] AND entradas.TR_L2_FT2_Tot.rtotal >= Total;
HMI.CA1_L2_V4_Cmd_Man R= _w10;
Liquidos.InyectarLiq[2] R= _w10;
Modo_Calibrar_L2 R= _w10;
auxIniCal R= _w10;
HMI.CmdM_PC1_L2_BD R= _w10;

// NETWORK 28
_w11 := auxIniCal AND Modo_Calibrar_L2 AND FALSE AND tInyeccion.Q;
HMI.CA1_L2_V4_Cmd_Man R= _w11;
Liquidos.InyectarLiq[2] R= _w11;
Modo_Calibrar_L2 R= _w11;
auxIniCal R= _w11;
HMI.CmdM_PC1_L2_BD R= _w11;

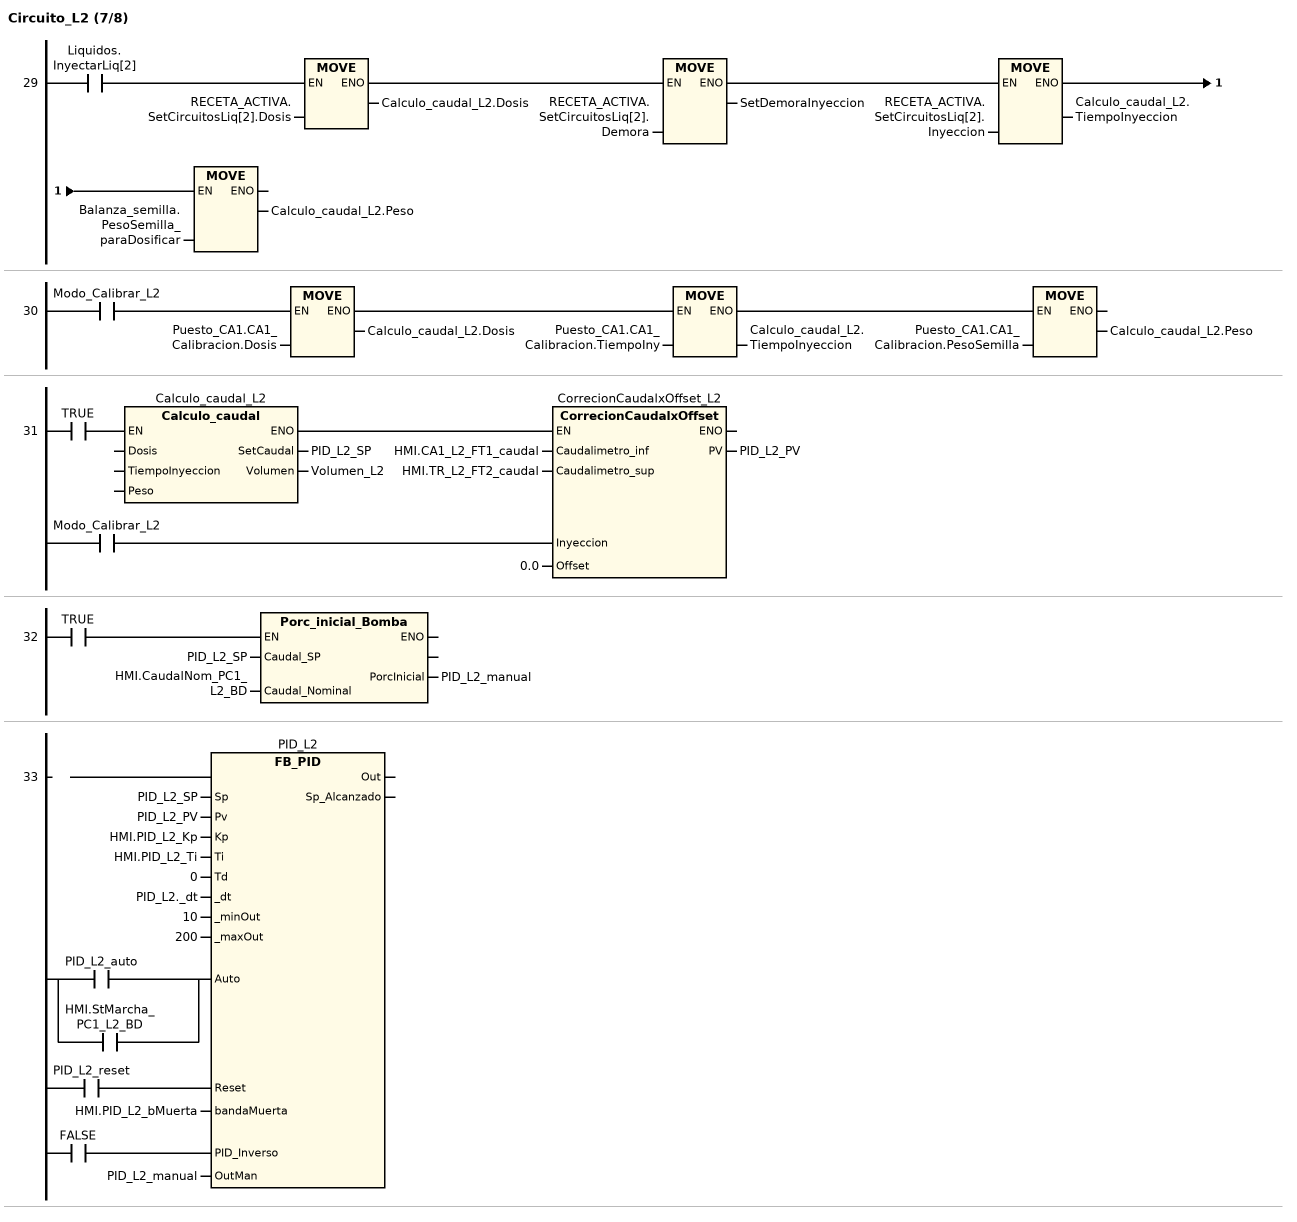
// NETWORK 29
_w12 := Liquidos.InyectarLiq[2];
IF _w12 THEN Calculo_caudal_L2.Dosis := RECETA_ACTIVA.SetCircuitosLiq[2].Dosis; END_IF
IF _w12 THEN SetDemoraInyeccion := RECETA_ACTIVA.SetCircuitosLiq[2].Demora; END_IF
IF _w12 THEN Calculo_caudal_L2.TiempoInyeccion := RECETA_ACTIVA.SetCircuitosLiq[2].Inyeccion; END_IF
IF _w12 THEN Calculo_caudal_L2.Peso := Balanza_semilla.PesoSemilla_paraDosificar; END_IF

// NETWORK 30
_w13 := Modo_Calibrar_L2;
IF _w13 THEN Calculo_caudal_L2.Dosis := Puesto_CA1.CA1_Calibracion.Dosis; END_IF
IF _w13 THEN Calculo_caudal_L2.TiempoInyeccion := Puesto_CA1.CA1_Calibracion.TiempoIny; END_IF
IF _w13 THEN Calculo_caudal_L2.Peso := Puesto_CA1.CA1_Calibracion.PesoSemilla; END_IF

// NETWORK 31
Calculo_caudal_L2(SetCaudal => PID_L2_SP, Volumen => Volumen_L2); // Calculo_caudal
CorrecionCaudalxOffset_L2(
    Caudalimetro_inf := HMI.CA1_L2_FT1_caudal,
    Caudalimetro_sup := HMI.TR_L2_FT2_caudal,
    Inyeccion := Modo_Calibrar_L2,
    Offset := 0.0,
    PV => PID_L2_PV); // CorrecionCaudalxOffset

// NETWORK 32
Porc_inicial_Bomba(Caudal_SP := PID_L2_SP, Caudal_Nominal := HMI.CaudalNom_PC1_L2_BD, PorcInicial => PID_L2_manual);

// NETWORK 33
PID_L2(
    Sp := PID_L2_SP,
    Pv := PID_L2_PV,
    Kp := HMI.PID_L2_Kp,
    Ti := HMI.PID_L2_Ti,
    Td := 0,
    _dt := PID_L2._dt,
    _minOut := 10,
    _maxOut := 200,
    Auto := PID_L2_auto OR HMI.StMarcha_PC1_L2_BD,
    Reset := PID_L2_reset,
    bandaMuerta := HMI.PID_L2_bMuerta,
    PID_Inverso := FALSE,
    OutMan := PID_L2_manual); // FB_PID

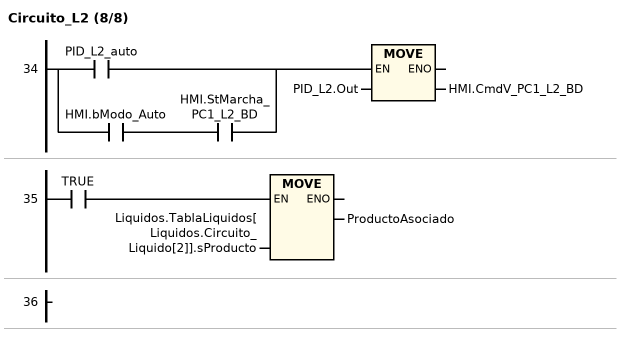
// NETWORK 34
IF PID_L2_auto OR HMI.bModo_Auto AND HMI.StMarcha_PC1_L2_BD THEN HMI.CmdV_PC1_L2_BD := PID_L2.Out; END_IF

// NETWORK 35
ProductoAsociado := Liquidos.TablaLiquidos[Liquidos.Circuito_Liquido[2]].sProducto;

// NETWORK 36

END_PROGRAM

// ---- POUs/Puesto_Calibracion_1/Puesto_CA1.TcPOU
PROGRAM Puesto_CA1
VAR
	Balanza_CA1: Balanza;
	dHS:DINT;
	Cmd_Full: R_TRIG;
	TmrLabelFinalizado: TON;
	CA1_Calibracion: Calibracion_Liq_calc;
	Tarar_balanza		:BOOL;
	Offset_ref			:REAL;
	Inyectar_ref		:BOOL;
	InicioCal_ref		:BOOL;
	PesoEspec			:REAL;
	UltimaCalibracao	:UDINT;
	VazaoMax			:REAL;

	Teste: BOOL;
END_VAR

VAR_INPUT
	// Vazão máxima da bomba excedida com esses parâmetros
	VazaoMaxExcedida: BOOL;
END_VAR

//Indica a ultima calibração da linha selecionada
UltimaCalibracao := HMI.UltimasCalibracoes[HMI.iCircuito_a_calibrar];

Balanza_CA1(
	wStatus:=Entradas.CA1_WT1_wStatus , 
	rValue_REAL:=Entradas.CA1_WT1_rValue_REAL , 
	nValue_DINT:=Entradas.CA1_WT1_nValue_DINT , 
	nValue_Supply:=dHS , 
	nValue_Bridge:=dHS , 
	stEcSlaveAmsNetAdr:=Entradas.CA1_WT1_stEcSlaveAmsNetAdr , 
	bWcState:=Entradas.CA1_WT1_bWcState , 
	wState:=Entradas.CA1_WT1_wState , 
	bCmd_FullCalibration:=HMI.bCmd_Full_WT_CA1 , 
	bCmd_ZeroCalibration:=HMI.bCmd_Zero_WT_CA1 , 
	bCmd_Tara:=Tarar_balanza , 
	bCmd_LoadReference:=HMI.bCmd_LoadReference_WT_CA1 ,
	fLoadReference:=(HMI.rPesoPatron_WT_CA1)/1000,
	wControl=>Salidas.CA1_WT1_wControl );
	
	TmrLabelFinalizado(IN:= HMI.bCmd_Full_WT_CA1 , PT:=T#10S , Q=> , ET=> );
	
	HMI.bCmd_LoadReference_WT_CA1:=FALSE;
	HMI.bCmd_Zero_WT_CA1:=FALSE;
	HMI.bCmd_Full_WT_CA1:=FALSE;
	Tarar_balanza:=FALSE;
	Cmd_Full(CLK:=TmrLabelFinalizado.Q , Q=> );
	IF 	Cmd_Full.Q THEN
		HMI.bCalibrado_WT_CA1:=TRUE;
	END_IF
/////////
PesoEspec:=Liquidos.TablaLiquidos[Liquidos.Circuito_Liquido[HMI.iCircuito_a_calibrar]].rDensidad;
CASE HMI.iCircuito_a_calibrar OF
	1:	Offset_ref:=Liquidos.Circuito_Offset[1];
		Inyectar_ref:=circuito_L1.Modo_Calibrar_L1;
		InicioCal_ref:=HMICA1.Inicio_calibracion;
		HMICA1.VolumenPedido_calibracion:=circuito_L1.Volumen_L1;
	2:	Offset_ref:=Liquidos.Circuito_Offset[2];
		Inyectar_ref:=circuito_L2.Modo_Calibrar_L2;
		InicioCal_ref:=HMICA1.Inicio_calibracion;
		HMICA1.VolumenPedido_calibracion:=circuito_L2.Volumen_L2;	
	3:	Offset_ref:=Liquidos.Circuito_Offset[3];
		Inyectar_ref:=circuito_L3.Modo_Calibrar_L3;
		InicioCal_ref:=HMICA1.Inicio_calibracion;
		HMICA1.VolumenPedido_calibracion:=circuito_L3.Volumen_L3;
	4:	Offset_ref:=Liquidos.Circuito_Offset[4];
		Inyectar_ref:=circuito_L4.Modo_Calibrar_L4;
		InicioCal_ref:=HMICA1.Inicio_calibracion;
		HMICA1.VolumenPedido_calibracion:=circuito_L4.Volumen_L4;	
		
		ELSE
	;		
END_CASE
	
/////////////////
CA1_Calibracion(
	Dosis:=HMICA1.Dosis_calibracion , 
	PesoSemilla:=HMICA1.Peso_calibracion,
	Tolerancia:=HMICA1.Tolerancia_calibracion , 
	PesoBalanza:=Entradas.CA1_WT1_rValue_REAL ,
	mlPedido:= HMICA1.VolumenPedido_calibracion,
	PesoEspec:=Puesto_CA1.PesoEspec , 
	Offset:=Offset_ref ,
	TiempoIny:=HMICA1.TInyeccion_calibracion , 
	Vol_Probeta:=(HMICA1.VolMaxProbeta_calibracion*1000) , 
	Pausa:=HMICA1.Pausa_calibracion , 
	Dosificar=> , 
	Probeta_Llena:=HMICA1.VaciarProbeta_calibracion , 
	Inyectar:=Inyectar_ref, 
	ml:=HMICA1.Volumen_calibracion, 
	Tiempo:=HMICA1.Tiempo_calibracion , 
	InicioCal:= InicioCal_ref, 
	Continuar:=HMICA1.Continuar_calibracion , 
	Tarar:=Tarar_balanza,
	Finalizado:=HMICA1.Fin_calibracion,
	mlProbeta=>HMICA1.Vol_enProbeta , 
	TiempoInyectado:=HMICA1.TiempoInyectado,
	Error_promedio=> HMICA1.Error_promedio, );
//
CASE HMI.iCircuito_a_calibrar OF
	1:	Liquidos.Circuito_Offset[1]:=Offset_ref;//Offset_ref
		circuito_L1.Modo_Calibrar_L1:=Inyectar_ref;//Inyectar_ref
		HMICA1.Inicio_calibracion:=InicioCal_ref;
		VazaoMax := HMI.CaudalNom_PC1_L1_BD;
	2:	Liquidos.Circuito_Offset[2]:=Offset_ref;//Offset_ref
		circuito_L2.Modo_Calibrar_L2:=Inyectar_ref;//Inyectar_ref
		HMICA1.Inicio_calibracion:=InicioCal_ref;
		VazaoMax := HMI.CaudalNom_PC1_L2_BD;
	3:	Liquidos.Circuito_Offset[3]:=Offset_ref;//Offset_refA
		circuito_L3.Modo_Calibrar_L3:=Inyectar_ref;//Inyectar_ref
		HMICA1.Inicio_calibracion:=InicioCal_ref;
		VazaoMax := HMI.CaudalNom_PC1_L3_BD;
	4:	Liquidos.Circuito_Offset[4]:=Offset_ref;//Offset_ref
		circuito_L4.Modo_Calibrar_L4:=Inyectar_ref;//Inyectar_ref
		HMICA1.Inicio_calibracion:=InicioCal_ref;
		VazaoMax := HMI.CaudalNom_PC1_L4_BD;
		
		ELSE
	;		
END_CASE

//Verifica se a vazão máxima suportada pela bomba foi excedida
IF HMICA1.TInyeccion_calibracion > 0 THEN
	IF (HMICA1.Dosis_calibracion*HMICA1.Peso_calibracion/100)/TO_REAL(HMICA1.TInyeccion_calibracion) > VazaoMax THEN
		VazaoMaxExcedida := TRUE;
	ELSE
		VazaoMaxExcedida := FALSE;
	END_IF
END_IF

END_PROGRAM

// ---- POUs/Elementos/Calibracion_Liq_calc.TcPOU
FUNCTION_BLOCK Calibracion_Liq_calc
VAR_INPUT
	Dosis :REAL;			//Dose a cada 100 kg
	PesoSemilla:REAL;		//Peso da batelada a ser tratada
	TiempoInyectado:DINT;	//Tempo de injeção
	Tolerancia:REAL;		//Tolerância ao erro
	PesoBalanza:REAL;
	PesoEspec:REAL;
	TiempoIny:DINT;
	Vol_Probeta:REAL;
	Pausa:BOOL;
	
END_VAR
VAR_OUTPUT
	Error_promedio:REAL;	//Erro médio
	Dosificar:BOOL;			//Fazer dosagem
	mlProbeta:REAL;

	
END_VAR
VAR_IN_OUT
	ml:ARRAY [1..3] OF REAL;
	Tiempo:ARRAY [1..3] OF DINT;
	InicioCal:BOOL;		
	Continuar:BOOL;
	Tarar:BOOL;
	mlPedido:REAL;		//mL que deve ter no recipiente ao final da injeção
	Offset	:REAL;
	Inyectar:BOOL;
	Probeta_Llena:BOOL;
	Finalizado:BOOL;
END_VAR
VAR
	Cant_cal_ok:INT;
	trigger:BOOL;
	posicion:INT;
	mlMedido:REAL;
	Aux_tiempo_iny:DINT;
	toleSup:REAL;	//Limite superior considerando o erro
	toleInf:REAL;	//Limite inferior considerando o erro
	sc_L:BOOL;
	aux_offset:REAL;
	aux_offset_correc:REAL;
	TON_3:TON;
	clock:BOOL;
	T_PesoBal:ARRAY [1..3] OF REAL;
	PesoBal:REAL;
	Prom_T_PesoBal:REAL;
	ET_clock:TIME;
	fbInicioCal:R_TRIG;

	Inyectando: BOOL;
	fbTmrCalculo:TON;
	fbCalcular:F_TRIG;
	Corregir:BOOL;
	fbTarar:TON;
	TaraOk:BOOL;
	Vol_enProbeta:REAL;
	Calcular:BOOL;
	bProbetaLlena:F_TRIG;
	bTaraOK:	F_TRIG;
	bInyectar: F_TRIG;
	bCalcular: R_TRIG;
	tarando: BOOL;
	Hug: BOOL;
	FinCalculo: BOOL;
	Calculando: BOOL;
	Step: INT;
	AuxVaciar: BOOL;
END_VAR
VAR PERSISTENT
	UltimaCalibracao	:UDINT;	//ùltima calibração feita com sucesso - Está como udint para correta conversão na IHM
END_VAR


IF InicioCal AND step=0 THEN
	Step:=1;
END_IF
IF NOT InicioCal  THEN
	Step:=0;
END_IF
CASE Step OF
	1:  //Inicializo variables y verifico valores peso semilla/dosis/tiempo inyeccion diferente de cero
		//Verificação se o peso da semente, a dose e tempo de injeção não 0, se for, são setados para 1
		IF PesoSemilla=0.0  THEN
			PesoSemilla:=1;
		END_IF
		IF Dosis=0.0  THEN
			Dosis:=1;
		END_IF
		IF TiempoIny=0  THEN
			TiempoIny:=1;
		END_IF
		mlPedido	:= Dosis*PesoSemilla/100;
		toleSup		:= mlPedido*(1.0+Tolerancia/100.0);
		toleInf		:= mlPedido*(1.0-Tolerancia/100.0);
		ml[1]		:= 0.0;
		ml[2]		:= 0.0;
		ml[3]		:= 0.0;
		Tiempo[1]	:= 0;
		Tiempo[2]	:= 0;
		Tiempo[3]	:= 0;
		mlProbeta	:= 0.0;
		Finalizado	:= 0;
		Tarar		:= TRUE;
		tarando		:= 1;
		Step		:= 2;
		
	2:  //
		bProbetaLlena(ClK:=Probeta_Llena,Q=>AuxVaciar);
		IF AuxVaciar THEN
			mlProbeta	:=0;
			AuxVaciar	:=0;
		END_IF
		IF NOT Probeta_Llena AND NOT Pausa THEN
			Tarar	:= InicioCal;
			tarando	:= InicioCal;
		END_IF
		fbTarar(IN:=(tarando),PT:=T#4S);
		//bProbetaLlena(ClK:=Probeta_Llena,Q=>AuxVaciar);
		//IF AuxVaciar THEN
		//	mlProbeta:=0;
		//	AuxVaciar:=0;
		//END_IF
		IF fbTarar.Q AND NOT Probeta_Llena AND NOT Pausa THEN
		tarando:=0;
		Inyectar:=1;
		Step:=3;
		END_IF
	3:	//espera de tiempo para realizar calculo de lo dosificado
		fbTmrCalculo (IN:=NOT Inyectar,PT:=T#6S);
		IF fbTmrCalculo.Q THEN
			Step:=4;
		END_IF
	4:	//calculo de los valores medidos
		IF PesoEspec <> 0 THEN
			mlMedido:=PesoBalanza/PesoEspec*1000;
		ELSE
			mlMedido := 0;
		END_IF
		
		mlProbeta:=mlProbeta+mlMedido;
		Aux_tiempo_iny:=TiempoInyectado;
		IF ((1.1*mlPedido+mlProbeta)>Vol_Probeta) THEN
			Probeta_Llena:=1;
		END_IF
	
		FOR posicion:=3 TO 2 BY -1 DO
			ml[posicion]:=ml[posicion-1];
			Tiempo[posicion]:=tiempo[posicion-1];
		END_FOR;
		ml[1]:=mlMedido;
		tiempo[1]:=Aux_tiempo_iny;
	
		IF ((mlMedido<toleInf) OR (mlMedido>toleSup)) THEN  //medicion fuera de tolerancia
			aux_offset:= SEL(mlPedido > 0, mlMedido , mlMedido/mlPedido);
			
			IF (aux_offset<=0.9) THEN
				aux_offset_correc:=0.06;
			END_IF;
			
			IF (aux_offset>0.9 AND aux_offset<0.95) THEN
				aux_offset_correc:=0.01;
			END_IF;	
			
			IF (aux_offset >= 0.95 AND aux_offset<1) THEN
				aux_offset_correc:=0.001;
			END_IF;	
		
			IF (aux_offset>1 AND aux_offset<1.05) THEN
				aux_offset_correc:=-0.001;
			END_IF;	
			
			IF (aux_offset>=1.05 AND aux_offset<1.1) THEN
				aux_offset_correc:=-0.01;
			END_IF;
			
			IF (aux_offset>=1.1) THEN
				aux_offset_correc:=-0.06;
			END_IF;
	
			Offset:=Offset+aux_offset_correc;
			Cant_cal_ok:=0;
			//Tarar:=InicioCal;
			//tarando:=InicioCal;
			Step:=2;
		ELSE
			Cant_cal_ok:=1+Cant_cal_ok;
			//Tarar:=InicioCal;
			//tarando:=InicioCal;
			Step:=2;
		END_IF
END_CASE


IF InicioCal AND Cant_cal_ok=3 THEN
	//Verifica a hora da ultima calibração e escreve na variável da linha em questão
	UltimaCalibracao := DT_TO_UDINT(MAIN.HoraAtual);
	HMI.UltimasCalibracoes[HMI.iCircuito_a_calibrar]	:= UltimaCalibracao;
	HMI.UltimoAlrCalibr[HMI.iCircuito_a_calibrar]		:= UltimaCalibracao;
	
	InicioCal	:=0;
	tarando		:=0;
	Finalizado	:=1;
	Error_promedio :=((ABS ( (ml[1]-mlPedido))+ABS ( (ml[2]-mlPedido))+ABS ( (ml[3]-mlPedido)))/(3.0*mlPedido))*100.0;
	Step	:=0;
END_IF

//reset valores finalizado
IF NOT InicioCal THEN
	Cant_cal_ok:=0;
	Vol_enProbeta:=0.0;
END_IF;

END_FUNCTION_BLOCK

// ---- POUs/Puesto_Calibracion_1/Circuito_L3.TcPOU
PROGRAM Circuito_L3
VAR_INPUT
			Modo_Calibrar_L3 :BOOL;
END_VAR
VAR
		fbBomba_L3 :Equipo_Motor_ATV320;
		Totalizador_L3: Totalizador;//totalizador caudalimetro inferior
		Totalizador_L3_s: Totalizador;//totalizador caudalimetro superior
		Reset_TotL3:BOOL;
		Reset_TotL3_s: BOOL;
		PID_L3:FB_PID;
		ControlValv_ioLink_V1:ControlValv_ioLink;
		ControlValv_ioLink_V2: ControlValv_ioLink;
		ControlValv_ioLink_V3: ControlValv_ioLink;
		ControlValv_ioLink_V4: ControlValv_ioLink;
		Falla_L3_V1:BOOL;
		Falla_L3_V2:BOOL;
		Falla_L3_V3:BOOL;
		Falla_L3_V4:BOOL;
		Balanza_PU1_WT3: Balanza;
		TOF_calibradoIBC: TOF;
		
		auxHS:BOOL;
		dHS:DINT;
		PID_L3_SP:REAL;
		PID_L3_auto:BOOL;
		PID_L3_reset:BOOL;
		PID_L3_manual:REAL;
		PID_L3_bMuerta:REAL := 5;
		PID_L3_Kp:REAL := 0.1;
		PID_L3_Ti:REAL := 100;
		PID_L3_PV:REAL;
		Dosis_L3	:REAL;
		TiempoInyeccion_L3	:DINT;
		Peso	:REAL;
		Offset_L3:REAL;
		Inyeccion_L3:BOOL;

		Volumen_L3:Real;
	Calculo_caudal_L3: Calculo_caudal;
	CorrecionCaudalxOffset_L3: CorrecionCaudalxOffset;
	tInyeccion: TON;
	Total :REAL;
	Totalant	:REAL;
	auxIniCal:BOOL;
	AuxVol:REAL;
	CA1_L3_V1_CmdA_Man :BOOL;
	CA1_L3_V4_CmdA_Man :BOOL;
	TDemoraInyectar: TON;
	SetDemoraInyeccion: REAL;
	TiempoDeInyeccion:TIME;
	Tiempo_TIME_to_seg_InyCal: Tiempo_TIME_to_seg;
	AuxInyCal:TIME;
	Tiempo_seg_to_TIME_DemoraInyec: Tiempo_seg_to_TIME;
	AuxTDemoraInyec: TIME;
	IniTotalFT2:REAL;
	Auxconsumo:REAL;
	ProductoAsociado: STRING;
	Lavagem_Circuito03: Lavagem;
	Filtro2_Teste: Filtro2;
	PID_GENERICO_0: PID_GENERICO;
END_VAR
VAR PERSISTENT
	UltimaCalibracao	:UDINT;	//Data e hora da ultima calibração
END_VAR
VAR // added by the converter: edge detectors and wires of the graphical bodies
    _w1, _w2, _w3, _w4, _w5, _w6, _w7, _w8, _w9, _w10, _w11, _w12, _w13 : BOOL;
    _ft1 : F_TRIG;
    _rt1, _rt2 : R_TRIG;
END_VAR

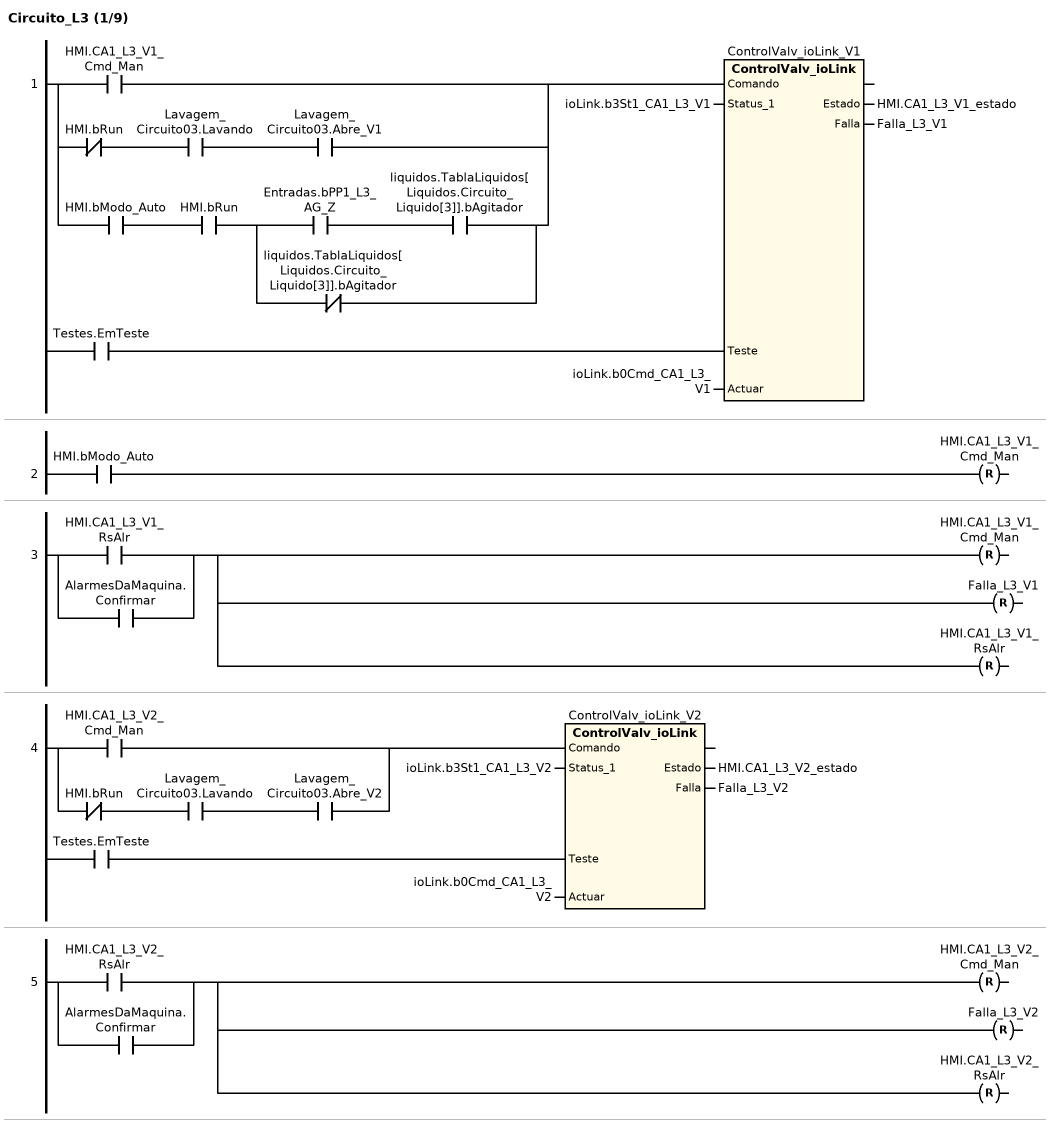
// NETWORK 1
ControlValv_ioLink_V1(
    Comando := HMI.CA1_L3_V1_Cmd_Man OR NOT HMI.bRun AND Lavagem_Circuito03.Lavando AND Lavagem_Circuito03.Abre_V1 OR HMI.bModo_Auto AND HMI.bRun AND (Entradas.bPP1_L3_AG_Z AND (liquidos.TablaLiquidos[Liquidos.Circuito_Liquido[3]].bAgitador) OR NOT (liquidos.TablaLiquidos[Liquidos.Circuito_Liquido[3]].bAgitador)),
    Status_1 := ioLink.b3St1_CA1_L3_V1,
    Teste := Testes.EmTeste,
    Actuar := ioLink.b0Cmd_CA1_L3_V1,
    Estado => HMI.CA1_L3_V1_estado,
    Falla => Falla_L3_V1); // ControlValv_ioLink

// NETWORK 2
HMI.CA1_L3_V1_Cmd_Man R= HMI.bModo_Auto;

// NETWORK 3
_w1 := HMI.CA1_L3_V1_RsAlr OR AlarmesDaMaquina.Confirmar;
HMI.CA1_L3_V1_Cmd_Man R= _w1;
Falla_L3_V1 R= _w1;
HMI.CA1_L3_V1_RsAlr R= _w1;

// NETWORK 4
ControlValv_ioLink_V2(
    Comando := HMI.CA1_L3_V2_Cmd_Man OR NOT HMI.bRun AND Lavagem_Circuito03.Lavando AND Lavagem_Circuito03.Abre_V2,
    Status_1 := ioLink.b3St1_CA1_L3_V2,
    Teste := Testes.EmTeste,
    Actuar := ioLink.b0Cmd_CA1_L3_V2,
    Estado => HMI.CA1_L3_V2_estado,
    Falla => Falla_L3_V2); // ControlValv_ioLink

// NETWORK 5
_w2 := HMI.CA1_L3_V2_RsAlr OR AlarmesDaMaquina.Confirmar;
HMI.CA1_L3_V2_Cmd_Man R= _w2;
Falla_L3_V2 R= _w2;
HMI.CA1_L3_V2_RsAlr R= _w2;

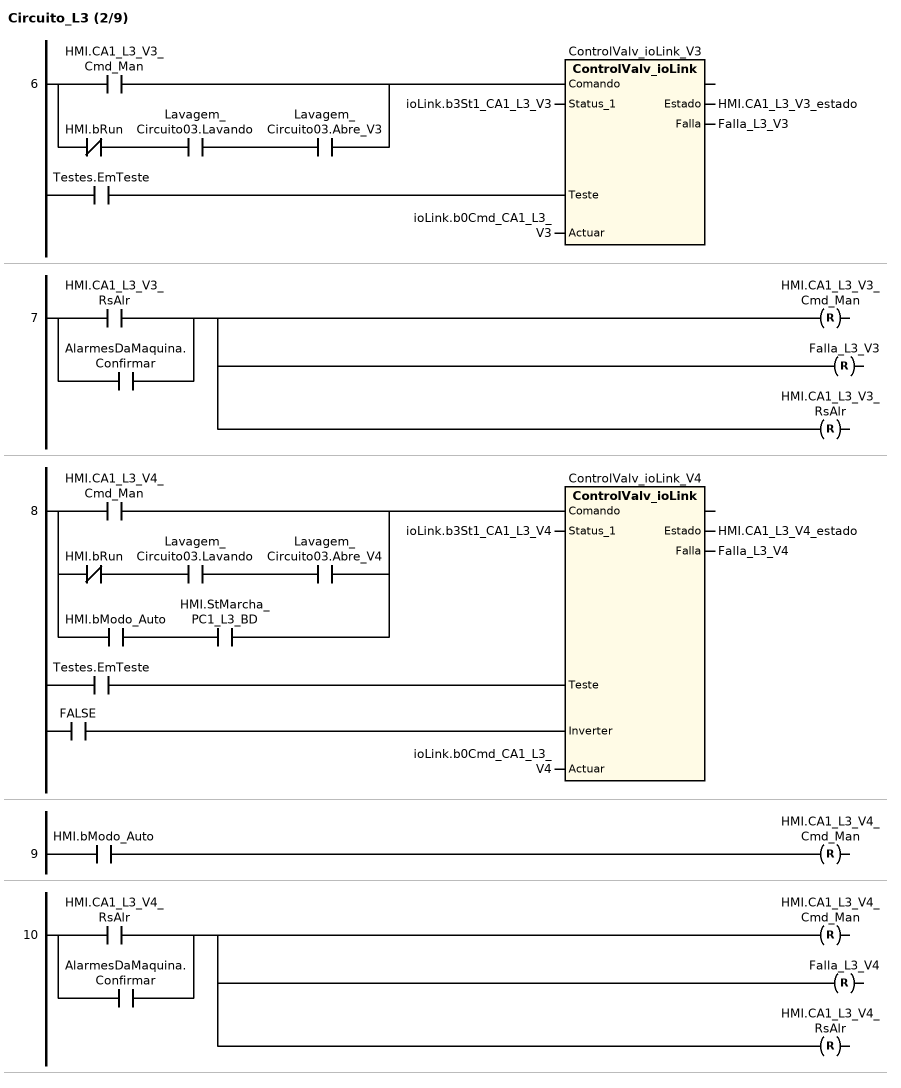
// NETWORK 6
ControlValv_ioLink_V3(
    Comando := HMI.CA1_L3_V3_Cmd_Man OR NOT HMI.bRun AND Lavagem_Circuito03.Lavando AND Lavagem_Circuito03.Abre_V3,
    Status_1 := ioLink.b3St1_CA1_L3_V3,
    Teste := Testes.EmTeste,
    Actuar := ioLink.b0Cmd_CA1_L3_V3,
    Estado => HMI.CA1_L3_V3_estado,
    Falla => Falla_L3_V3); // ControlValv_ioLink

// NETWORK 7
_w3 := HMI.CA1_L3_V3_RsAlr OR AlarmesDaMaquina.Confirmar;
HMI.CA1_L3_V3_Cmd_Man R= _w3;
Falla_L3_V3 R= _w3;
HMI.CA1_L3_V3_RsAlr R= _w3;

// NETWORK 8
ControlValv_ioLink_V4(
    Comando := HMI.CA1_L3_V4_Cmd_Man OR NOT HMI.bRun AND Lavagem_Circuito03.Lavando AND Lavagem_Circuito03.Abre_V4 OR HMI.bModo_Auto AND HMI.StMarcha_PC1_L3_BD,
    Status_1 := ioLink.b3St1_CA1_L3_V4,
    Teste := Testes.EmTeste,
    Inverter := FALSE,
    Actuar := ioLink.b0Cmd_CA1_L3_V4,
    Estado => HMI.CA1_L3_V4_estado,
    Falla => Falla_L3_V4); // ControlValv_ioLink

// NETWORK 9
HMI.CA1_L3_V4_Cmd_Man R= HMI.bModo_Auto;

// NETWORK 10
_w4 := HMI.CA1_L3_V4_RsAlr OR AlarmesDaMaquina.Confirmar;
HMI.CA1_L3_V4_Cmd_Man R= _w4;
Falla_L3_V4 R= _w4;
HMI.CA1_L3_V4_RsAlr R= _w4;

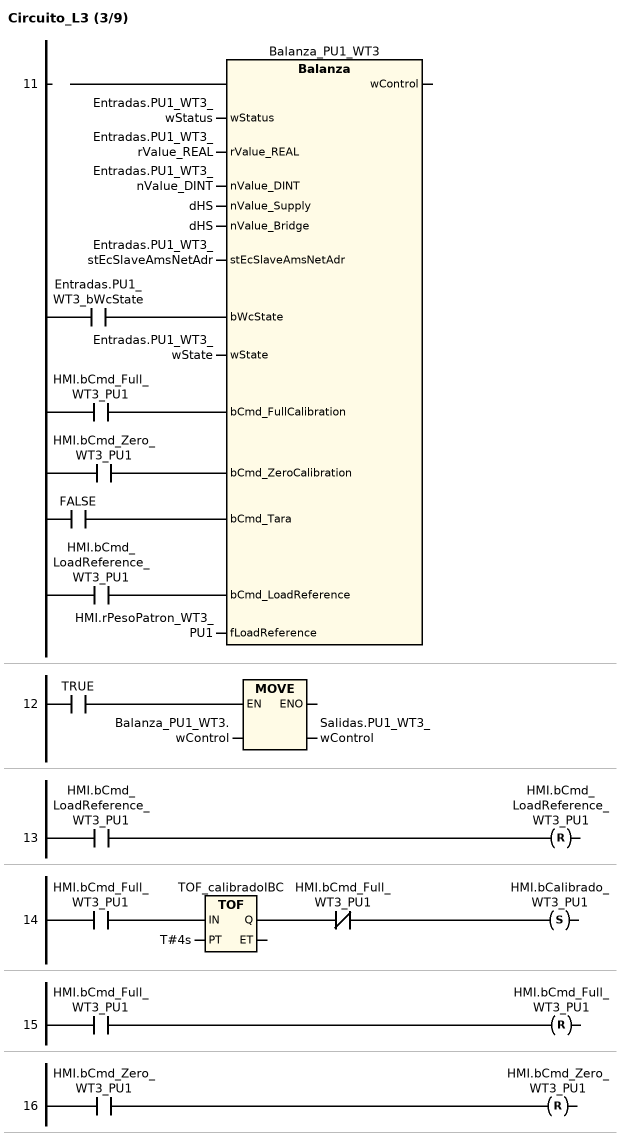
// NETWORK 11
Balanza_PU1_WT3(
    wStatus := Entradas.PU1_WT3_wStatus,
    rValue_REAL := Entradas.PU1_WT3_rValue_REAL,
    nValue_DINT := Entradas.PU1_WT3_nValue_DINT,
    nValue_Supply := dHS,
    nValue_Bridge := dHS,
    stEcSlaveAmsNetAdr := Entradas.PU1_WT3_stEcSlaveAmsNetAdr,
    bWcState := Entradas.PU1_WT3_bWcState,
    wState := Entradas.PU1_WT3_wState,
    bCmd_FullCalibration := HMI.bCmd_Full_WT3_PU1,
    bCmd_ZeroCalibration := HMI.bCmd_Zero_WT3_PU1,
    bCmd_Tara := FALSE,
    bCmd_LoadReference := HMI.bCmd_LoadReference_WT3_PU1,
    fLoadReference := HMI.rPesoPatron_WT3_PU1); // Balanza

// NETWORK 12
Salidas.PU1_WT3_wControl := Balanza_PU1_WT3.wControl;

// NETWORK 13
HMI.bCmd_LoadReference_WT3_PU1 R= HMI.bCmd_LoadReference_WT3_PU1;

// NETWORK 14
TOF_calibradoIBC(IN := HMI.bCmd_Full_WT3_PU1, PT := T#4s); // TOF
HMI.bCalibrado_WT3_PU1 S= TOF_calibradoIBC.Q AND NOT HMI.bCmd_Full_WT3_PU1;

// NETWORK 15
HMI.bCmd_Full_WT3_PU1 R= HMI.bCmd_Full_WT3_PU1;

// NETWORK 16
HMI.bCmd_Zero_WT3_PU1 R= HMI.bCmd_Zero_WT3_PU1;

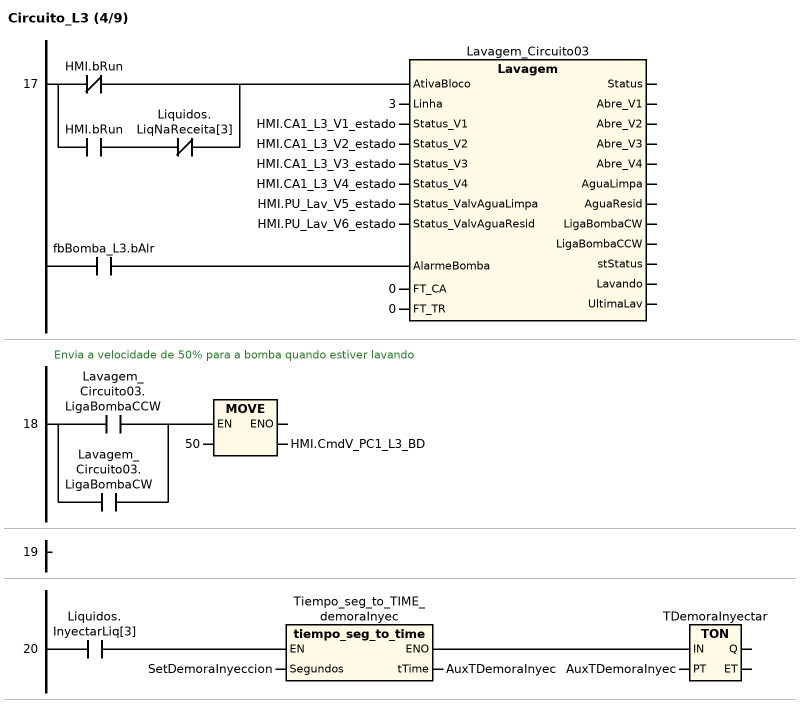
// NETWORK 17
Lavagem_Circuito03(
    AtivaBloco := NOT HMI.bRun OR HMI.bRun AND NOT Liquidos.LiqNaReceita[3],
    Linha := 3,
    Status_V1 := HMI.CA1_L3_V1_estado,
    Status_V2 := HMI.CA1_L3_V2_estado,
    Status_V3 := HMI.CA1_L3_V3_estado,
    Status_V4 := HMI.CA1_L3_V4_estado,
    Status_ValvAguaLimpa := HMI.PU_Lav_V5_estado,
    Status_ValvAguaResid := HMI.PU_Lav_V6_estado,
    AlarmeBomba := fbBomba_L3.bAlr,
    FT_CA := 0,
    FT_TR := 0); // Lavagem

// NETWORK 18
// Envia a velocidade de 50% para a bomba quando estiver lavando
IF Lavagem_Circuito03.LigaBombaCCW OR Lavagem_Circuito03.LigaBombaCW THEN HMI.CmdV_PC1_L3_BD := 50; END_IF

// NETWORK 19

// NETWORK 20
_w5 := Liquidos.InyectarLiq[3];
IF _w5 THEN
    Tiempo_seg_to_TIME_demoraInyec(Segundos := SetDemoraInyeccion, tTime => AuxTDemoraInyec); // tiempo_seg_to_time
END_IF
TDemoraInyectar(IN := _w5, PT := AuxTDemoraInyec); // TON

